ABB RAPID module: ecde059d.mod

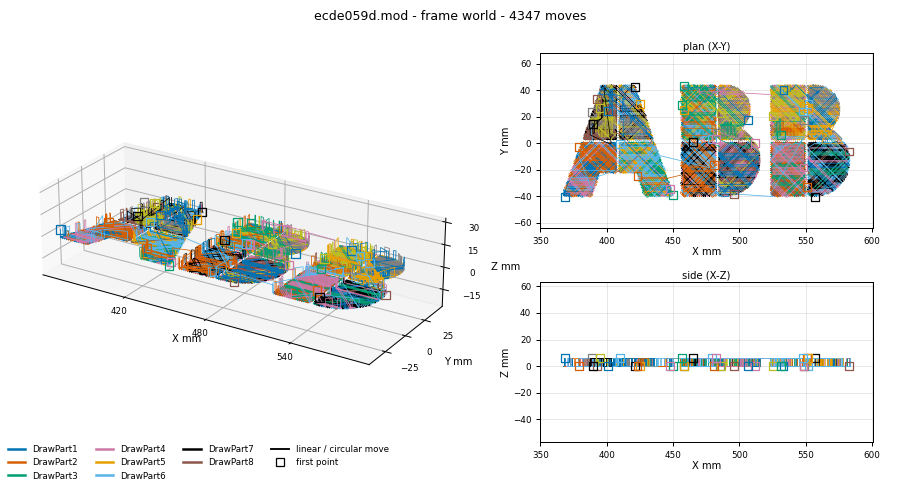
[picture p0: tool path of ecde059d.mod in frame world, 4347 of 4349 moves have a stored position in this frame; points joined in program order, loops and branches not executed]
MODULE ImageDraw
  ! Generated 2026-10-07 06:31 for ABB GoFa CRB 15000-5/0.95: 465 strokes
  ! Page 250 x 180 mm. Work object wPaper: Z points up, so pen-up is +Z and the tool uses orientation [0,1,0,0].
  PERS tooldata tPen:=[TRUE,[[0,0,120],[1,0,0,0]],[0.3,[0,0,60],[1,0,0,0],0,0,0]];
  PERS wobjdata wPaper:=[FALSE,TRUE,"",[[350,-90,0],[1,0,0,0]],[[0,0,0],[1,0,0,0]]];
  CONST robtarget pOrigin:=[[0,0,0],[0,1,0,0],[0,0,0,0],[9E9,9E9,9E9,9E9,9E9,9E9]];
  CONST jointtarget jHome:=[[0,0,0,0,30,0],[9E9,9E9,9E9,9E9,9E9,9E9]];
  CONST speeddata vTravel:=[250,200,5000,1000];

  PROC DrawImage()
    SingArea\Wrist;
    ConfL\Off;
    ConfJ\Off;
    MoveAbsJ jHome\NoEOffs,vTravel,fine,tPen;
    DrawPart1;
    DrawPart2;
    DrawPart3;
    DrawPart4;
    DrawPart5;
    DrawPart6;
    DrawPart7;
    DrawPart8;
    DrawPart9;
    DrawPart10;
    DrawPart11;
    DrawPart12;
    DrawPart13;
    DrawPart14;
    DrawPart15;
    DrawPart16;
    DrawPart17;
    DrawPart18;
    DrawPart19;
    DrawPart20;
    DrawPart21;
    DrawPart22;
    DrawPart23;
    DrawPart24;
    DrawPart25;
    DrawPart26;
    DrawPart27;
    DrawPart28;
    DrawPart29;
    DrawPart30;
    DrawPart31;
    DrawPart32;
    DrawPart33;
    DrawPart34;
    DrawPart35;
    DrawPart36;
    DrawPart37;
    MoveAbsJ jHome\NoEOffs,vTravel,fine,tPen;
  ENDPROC

  PROC DrawPart1()
    MoveL Offs(pOrigin,18.68,49.65,6.00),vTravel,z5,tPen\WObj:=wPaper;
    MoveL Offs(pOrigin,18.68,49.65,0.00),v60,z0,tPen\WObj:=wPaper;
    MoveL Offs(pOrigin,16.98,51.35,0.00),v40,z0,tPen\WObj:=wPaper;
    MoveL Offs(pOrigin,17.75,50.83,0.00),v40,z0,tPen\WObj:=wPaper;
    MoveL Offs(pOrigin,38.15,50.83,0.00),v40,z0,tPen\WObj:=wPaper;
    MoveL Offs(pOrigin,44.15,68.12,0.00),v40,z0,tPen\WObj:=wPaper;
    MoveL Offs(pOrigin,57.05,68.32,0.00),v40,z0,tPen\WObj:=wPaper;
    MoveL Offs(pOrigin,57.05,90.47,0.00),v40,z0,tPen\WObj:=wPaper;
    MoveL Offs(pOrigin,31.55,90.38,0.00),v40,z0,tPen\WObj:=wPaper;
    MoveL Offs(pOrigin,17.80,51.83,0.00),v40,z0,tPen\WObj:=wPaper;
    MoveL Offs(pOrigin,17.75,50.83,0.00),v40,z0,tPen\WObj:=wPaper;
    MoveL Offs(pOrigin,18.37,50.89,0.00),v40,z0,tPen\WObj:=wPaper;
    MoveL Offs(pOrigin,56.88,89.39,0.00),v40,z0,tPen\WObj:=wPaper;
    MoveL Offs(pOrigin,56.13,90.14,0.00),v40,z0,tPen\WObj:=wPaper;
    MoveL Offs(pOrigin,17.84,51.85,0.00),v40,z0,tPen\WObj:=wPaper;
    MoveL Offs(pOrigin,17.20,52.63,0.00),v40,z0,tPen\WObj:=wPaper;
    MoveL Offs(pOrigin,20.06,49.76,0.00),v40,z0,tPen\WObj:=wPaper;
    MoveL Offs(pOrigin,19.65,50.67,0.00),v40,z0,tPen\WObj:=wPaper;
    MoveL Offs(pOrigin,56.88,87.90,0.00),v40,z0,tPen\WObj:=wPaper;
    MoveL Offs(pOrigin,56.15,87.51,0.00),v40,z0,tPen\WObj:=wPaper;
    MoveL Offs(pOrigin,31.55,87.51,0.00),v40,z0,tPen\WObj:=wPaper;
    MoveL Offs(pOrigin,31.70,88.57,0.00),v40,z0,tPen\WObj:=wPaper;
    MoveL Offs(pOrigin,56.15,88.57,0.00),v40,fine,tPen\WObj:=wPaper;
    MoveL Offs(pOrigin,56.15,88.57,6.00),v60,z5,tPen\WObj:=wPaper;
    MoveL Offs(pOrigin,57.51,88.48,6.00),vTravel,z5,tPen\WObj:=wPaper;
    MoveL Offs(pOrigin,57.51,88.48,0.00),v60,z0,tPen\WObj:=wPaper;
    MoveL Offs(pOrigin,55.17,90.81,0.00),v40,z0,tPen\WObj:=wPaper;
    MoveL Offs(pOrigin,54.75,90.25,0.00),v40,z0,tPen\WObj:=wPaper;
    MoveL Offs(pOrigin,18.47,53.98,0.00),v40,z0,tPen\WObj:=wPaper;
    MoveL Offs(pOrigin,19.40,53.72,0.00),v40,z0,tPen\WObj:=wPaper;
    MoveL Offs(pOrigin,38.30,53.72,0.00),v40,z0,tPen\WObj:=wPaper;
    MoveL Offs(pOrigin,39.32,53.92,0.00),v40,z0,tPen\WObj:=wPaper;
    MoveL Offs(pOrigin,36.14,50.73,0.00),v40,fine,tPen\WObj:=wPaper;
    MoveL Offs(pOrigin,36.14,50.73,6.00),v60,z5,tPen\WObj:=wPaper;
    MoveL Offs(pOrigin,34.75,50.84,6.00),vTravel,z5,tPen\WObj:=wPaper;
    MoveL Offs(pOrigin,34.75,50.84,0.00),v60,z0,tPen\WObj:=wPaper;
    MoveL Offs(pOrigin,39.85,55.94,0.00),v40,z0,tPen\WObj:=wPaper;
    MoveL Offs(pOrigin,39.05,55.83,0.00),v40,z0,tPen\WObj:=wPaper;
    MoveL Offs(pOrigin,20.15,55.83,0.00),v40,z0,tPen\WObj:=wPaper;
    MoveL Offs(pOrigin,19.21,56.21,0.00),v40,z0,tPen\WObj:=wPaper;
    MoveL Offs(pOrigin,53.47,90.47,0.00),v40,z0,tPen\WObj:=wPaper;
    MoveL Offs(pOrigin,53.58,90.92,0.00),v40,z0,tPen\WObj:=wPaper;
    MoveL Offs(pOrigin,57.50,86.99,0.00),v40,z0,tPen\WObj:=wPaper;
    MoveL Offs(pOrigin,56.88,86.41,0.00),v40,z0,tPen\WObj:=wPaper;
    MoveL Offs(pOrigin,21.25,50.78,0.00),v40,z0,tPen\WObj:=wPaper;
    MoveL Offs(pOrigin,21.55,49.77,0.00),v40,z0,tPen\WObj:=wPaper;
    MoveL Offs(pOrigin,17.42,53.90,0.00),v40,fine,tPen\WObj:=wPaper;
    MoveL Offs(pOrigin,17.42,53.90,6.00),v60,z5,tPen\WObj:=wPaper;
    MoveL Offs(pOrigin,17.53,55.29,6.00),vTravel,z5,tPen\WObj:=wPaper;
    MoveL Offs(pOrigin,17.53,55.29,0.00),v60,z0,tPen\WObj:=wPaper;
    MoveL Offs(pOrigin,23.47,49.35,0.00),v40,fine,tPen\WObj:=wPaper;
    MoveL Offs(pOrigin,23.47,49.35,6.00),v60,z5,tPen\WObj:=wPaper;
    MoveL Offs(pOrigin,24.12,50.66,6.00),vTravel,z5,tPen\WObj:=wPaper;
    MoveL Offs(pOrigin,24.12,50.66,0.00),v60,z0,tPen\WObj:=wPaper;
    MoveL Offs(pOrigin,56.89,83.44,0.00),v40,z0,tPen\WObj:=wPaper;
    MoveL Offs(pOrigin,57.60,83.91,0.00),v40,z0,tPen\WObj:=wPaper;
    MoveL Offs(pOrigin,50.71,90.80,0.00),v40,z0,tPen\WObj:=wPaper;
    MoveL Offs(pOrigin,50.28,90.26,0.00),v40,z0,tPen\WObj:=wPaper;
    MoveL Offs(pOrigin,20.79,60.78,0.00),v40,z0,tPen\WObj:=wPaper;
    MoveL Offs(pOrigin,20.31,61.46,0.00),v40,z0,tPen\WObj:=wPaper;
    MoveL Offs(pOrigin,32.29,49.48,0.00),v40,fine,tPen\WObj:=wPaper;
    MoveL Offs(pOrigin,32.29,49.48,6.00),v60,z5,tPen\WObj:=wPaper;
    MoveL Offs(pOrigin,31.02,49.26,6.00),vTravel,z5,tPen\WObj:=wPaper;
    MoveL Offs(pOrigin,31.02,49.26,0.00),v60,z0,tPen\WObj:=wPaper;
    MoveL Offs(pOrigin,19.77,60.51,0.00),v40,z0,tPen\WObj:=wPaper;
    MoveL Offs(pOrigin,19.35,59.44,0.00),v40,z0,tPen\WObj:=wPaper;
    MoveL Offs(pOrigin,29.10,49.68,0.00),v40,z0,tPen\WObj:=wPaper;
    MoveL Offs(pOrigin,28.59,50.65,0.00),v40,z0,tPen\WObj:=wPaper;
    MoveL Offs(pOrigin,43.12,65.18,0.00),v40,z0,tPen\WObj:=wPaper;
    MoveL Offs(pOrigin,42.35,65.34,0.00),v40,z0,tPen\WObj:=wPaper;
    MoveL Offs(pOrigin,23.60,65.34,0.00),v40,z0,tPen\WObj:=wPaper;
    MoveL Offs(pOrigin,23.90,66.39,0.00),v40,z0,tPen\WObj:=wPaper;
    MoveL Offs(pOrigin,42.65,66.39,0.00),v40,z0,tPen\WObj:=wPaper;
    MoveL Offs(pOrigin,42.95,67.45,0.00),v40,z0,tPen\WObj:=wPaper;
    MoveL Offs(pOrigin,24.35,67.45,0.00),v40,z0,tPen\WObj:=wPaper;
    MoveL Offs(pOrigin,24.65,68.50,0.00),v40,z0,tPen\WObj:=wPaper;
    MoveL Offs(pOrigin,43.85,68.50,0.00),v40,fine,tPen\WObj:=wPaper;
    MoveL Offs(pOrigin,43.85,68.50,6.00),v60,z5,tPen\WObj:=wPaper;
    MoveL Offs(pOrigin,44.58,67.06,6.00),vTravel,z5,tPen\WObj:=wPaper;
    MoveL Offs(pOrigin,44.58,67.06,0.00),v60,z0,tPen\WObj:=wPaper;
    MoveL Offs(pOrigin,28.35,83.29,0.00),v40,z0,tPen\WObj:=wPaper;
    MoveL Offs(pOrigin,27.92,82.23,0.00),v40,z0,tPen\WObj:=wPaper;
    MoveL Offs(pOrigin,44.15,66.00,0.00),v40,fine,tPen\WObj:=wPaper;
    MoveL Offs(pOrigin,44.15,66.00,6.00),v60,z5,tPen\WObj:=wPaper;
    MoveL Offs(pOrigin,43.83,64.83,6.00),vTravel,z5,tPen\WObj:=wPaper;
    MoveL Offs(pOrigin,43.83,64.83,0.00),v60,z0,tPen\WObj:=wPaper;
    MoveL Offs(pOrigin,27.28,81.37,0.00),v40,z0,tPen\WObj:=wPaper;
    MoveL Offs(pOrigin,26.85,80.31,0.00),v40,z0,tPen\WObj:=wPaper;
    MoveL Offs(pOrigin,43.50,63.66,0.00),v40,z0,tPen\WObj:=wPaper;
    MoveL Offs(pOrigin,43.07,62.59,0.00),v40,z0,tPen\WObj:=wPaper;
    MoveL Offs(pOrigin,26.53,79.14,0.00),v40,z0,tPen\WObj:=wPaper;
    MoveL Offs(pOrigin,27.44,79.37,0.00),v40,z0,tPen\WObj:=wPaper;
    MoveL Offs(pOrigin,38.58,90.51,0.00),v40,z0,tPen\WObj:=wPaper;
    MoveL Offs(pOrigin,38.37,91.19,0.00),v40,z0,tPen\WObj:=wPaper;
    MoveL Offs(pOrigin,57.78,71.78,0.00),v40,z0,tPen\WObj:=wPaper;
    MoveL Offs(pOrigin,57.03,71.63,0.00),v40,z0,tPen\WObj:=wPaper;
    MoveL Offs(pOrigin,53.64,68.24,0.00),v40,z0,tPen\WObj:=wPaper;
    MoveL Offs(pOrigin,53.19,67.41,0.00),v40,z0,tPen\WObj:=wPaper;
    MoveL Offs(pOrigin,30.50,90.11,0.00),v40,z0,tPen\WObj:=wPaper;
    MoveL Offs(pOrigin,31.24,90.85,0.00),v40,z0,tPen\WObj:=wPaper;
    MoveL Offs(pOrigin,55.11,66.99,0.00),v40,fine,tPen\WObj:=wPaper;
    MoveL Offs(pOrigin,55.11,66.99,6.00),v60,z5,tPen\WObj:=wPaper;
    MoveL Offs(pOrigin,55.13,68.23,6.00),vTravel,z5,tPen\WObj:=wPaper;
    MoveL Offs(pOrigin,55.13,68.23,0.00),v60,z0,tPen\WObj:=wPaper;
    MoveL Offs(pOrigin,57.04,70.14,0.00),v40,z0,tPen\WObj:=wPaper;
    MoveL Offs(pOrigin,56.15,70.62,0.00),v40,z0,tPen\WObj:=wPaper;
    MoveL Offs(pOrigin,25.40,70.62,0.00),v40,z0,tPen\WObj:=wPaper;
    MoveL Offs(pOrigin,25.85,71.67,0.00),v40,z0,tPen\WObj:=wPaper;
    MoveL Offs(pOrigin,56.15,71.67,0.00),v40,z0,tPen\WObj:=wPaper;
    MoveL Offs(pOrigin,56.15,72.73,0.00),v40,z0,tPen\WObj:=wPaper;
    MoveL Offs(pOrigin,26.30,72.73,0.00),v40,z0,tPen\WObj:=wPaper;
    MoveL Offs(pOrigin,26.60,73.78,0.00),v40,z0,tPen\WObj:=wPaper;
    MoveL Offs(pOrigin,56.15,73.78,0.00),v40,z0,tPen\WObj:=wPaper;
    MoveL Offs(pOrigin,56.15,74.84,0.00),v40,z0,tPen\WObj:=wPaper;
    MoveL Offs(pOrigin,27.05,74.84,0.00),v40,z0,tPen\WObj:=wPaper;
    MoveL Offs(pOrigin,27.50,75.90,0.00),v40,z0,tPen\WObj:=wPaper;
    MoveL Offs(pOrigin,56.00,75.90,0.00),v40,z0,tPen\WObj:=wPaper;
    MoveL Offs(pOrigin,56.81,75.88,0.00),v40,z0,tPen\WObj:=wPaper;
    MoveL Offs(pOrigin,49.17,68.25,0.00),v40,z0,tPen\WObj:=wPaper;
    MoveL Offs(pOrigin,49.04,67.08,0.00),v40,z0,tPen\WObj:=wPaper;
  ENDPROC

  PROC DrawPart2()
    MoveL Offs(pOrigin,29.32,86.81,0.00),v40,z0,tPen\WObj:=wPaper;
    MoveL Offs(pOrigin,29.97,86.39,0.00),v40,z0,tPen\WObj:=wPaper;
    MoveL Offs(pOrigin,34.11,90.52,0.00),v40,z0,tPen\WObj:=wPaper;
    MoveL Offs(pOrigin,34.22,90.86,0.00),v40,z0,tPen\WObj:=wPaper;
    MoveL Offs(pOrigin,57.24,67.84,0.00),v40,z0,tPen\WObj:=wPaper;
    MoveL Offs(pOrigin,56.38,67.20,0.00),v40,z0,tPen\WObj:=wPaper;
    MoveL Offs(pOrigin,32.41,91.18,0.00),v40,z0,tPen\WObj:=wPaper;
    MoveL Offs(pOrigin,32.62,90.53,0.00),v40,z0,tPen\WObj:=wPaper;
    MoveL Offs(pOrigin,30.82,88.72,0.00),v40,z0,tPen\WObj:=wPaper;
    MoveL Offs(pOrigin,30.17,88.94,0.00),v40,z0,tPen\WObj:=wPaper;
    MoveL Offs(pOrigin,51.70,67.40,0.00),v40,z0,tPen\WObj:=wPaper;
    MoveL Offs(pOrigin,52.26,68.35,0.00),v40,z0,tPen\WObj:=wPaper;
    MoveL Offs(pOrigin,57.03,73.12,0.00),v40,z0,tPen\WObj:=wPaper;
    MoveL Offs(pOrigin,57.78,73.27,0.00),v40,z0,tPen\WObj:=wPaper;
    MoveL Offs(pOrigin,40.18,90.88,0.00),v40,z0,tPen\WObj:=wPaper;
    MoveL Offs(pOrigin,40.07,90.50,0.00),v40,z0,tPen\WObj:=wPaper;
    MoveL Offs(pOrigin,26.81,77.25,0.00),v40,z0,tPen\WObj:=wPaper;
    MoveL Offs(pOrigin,27.80,76.95,0.00),v40,z0,tPen\WObj:=wPaper;
    MoveL Offs(pOrigin,56.00,76.95,0.00),v40,z0,tPen\WObj:=wPaper;
    MoveL Offs(pOrigin,56.80,77.37,0.00),v40,z0,tPen\WObj:=wPaper;
    MoveL Offs(pOrigin,47.68,68.25,0.00),v40,z0,tPen\WObj:=wPaper;
    MoveL Offs(pOrigin,47.34,67.28,0.00),v40,z0,tPen\WObj:=wPaper;
    MoveL Offs(pOrigin,28.99,85.63,0.00),v40,fine,tPen\WObj:=wPaper;
    MoveL Offs(pOrigin,28.99,85.63,6.00),v60,z5,tPen\WObj:=wPaper;
    MoveL Offs(pOrigin,28.67,84.46,6.00),vTravel,z5,tPen\WObj:=wPaper;
    MoveL Offs(pOrigin,28.67,84.46,0.00),v60,z0,tPen\WObj:=wPaper;
    MoveL Offs(pOrigin,45.75,67.39,0.00),v40,z0,tPen\WObj:=wPaper;
    MoveL Offs(pOrigin,46.19,68.26,0.00),v40,z0,tPen\WObj:=wPaper;
    MoveL Offs(pOrigin,56.91,78.97,0.00),v40,z0,tPen\WObj:=wPaper;
    MoveL Offs(pOrigin,57.48,79.55,0.00),v40,z0,tPen\WObj:=wPaper;
    MoveL Offs(pOrigin,46.13,90.90,0.00),v40,z0,tPen\WObj:=wPaper;
    MoveL Offs(pOrigin,46.02,90.49,0.00),v40,z0,tPen\WObj:=wPaper;
    MoveL Offs(pOrigin,23.22,67.68,0.00),v40,z0,tPen\WObj:=wPaper;
    MoveL Offs(pOrigin,22.46,68.28,0.00),v40,z0,tPen\WObj:=wPaper;
    MoveL Offs(pOrigin,39.43,51.31,0.00),v40,z0,tPen\WObj:=wPaper;
    MoveL Offs(pOrigin,38.89,50.35,0.00),v40,z0,tPen\WObj:=wPaper;
    MoveL Offs(pOrigin,22.03,67.21,0.00),v40,z0,tPen\WObj:=wPaper;
    MoveL Offs(pOrigin,21.49,66.25,0.00),v40,z0,tPen\WObj:=wPaper;
    MoveL Offs(pOrigin,38.25,49.50,0.00),v40,fine,tPen\WObj:=wPaper;
    MoveL Offs(pOrigin,38.25,49.50,6.00),v60,z5,tPen\WObj:=wPaper;
    MoveL Offs(pOrigin,36.76,49.49,6.00),vTravel,z5,tPen\WObj:=wPaper;
    MoveL Offs(pOrigin,36.76,49.49,0.00),v60,z0,tPen\WObj:=wPaper;
    MoveL Offs(pOrigin,21.06,65.19,0.00),v40,fine,tPen\WObj:=wPaper;
    MoveL Offs(pOrigin,21.06,65.19,6.00),v60,z5,tPen\WObj:=wPaper;
    MoveL Offs(pOrigin,22.27,65.24,6.00),vTravel,z5,tPen\WObj:=wPaper;
    MoveL Offs(pOrigin,22.27,65.24,0.00),v60,z0,tPen\WObj:=wPaper;
    MoveL Offs(pOrigin,47.30,90.27,0.00),v40,z0,tPen\WObj:=wPaper;
    MoveL Offs(pOrigin,47.73,90.79,0.00),v40,z0,tPen\WObj:=wPaper;
    MoveL Offs(pOrigin,57.49,81.04,0.00),v40,z0,tPen\WObj:=wPaper;
    MoveL Offs(pOrigin,56.90,80.46,0.00),v40,z0,tPen\WObj:=wPaper;
    MoveL Offs(pOrigin,27.10,50.65,0.00),v40,z0,tPen\WObj:=wPaper;
    MoveL Offs(pOrigin,27.51,49.78,0.00),v40,z0,tPen\WObj:=wPaper;
    MoveL Offs(pOrigin,19.02,58.27,0.00),v40,z0,tPen\WObj:=wPaper;
    MoveL Offs(pOrigin,19.95,58.44,0.00),v40,z0,tPen\WObj:=wPaper;
    MoveL Offs(pOrigin,51.98,90.47,0.00),v40,z0,tPen\WObj:=wPaper;
    MoveL Offs(pOrigin,52.09,90.91,0.00),v40,z0,tPen\WObj:=wPaper;
    MoveL Offs(pOrigin,57.50,85.50,0.00),v40,z0,tPen\WObj:=wPaper;
    MoveL Offs(pOrigin,56.89,84.93,0.00),v40,z0,tPen\WObj:=wPaper;
    MoveL Offs(pOrigin,22.63,50.67,0.00),v40,fine,tPen\WObj:=wPaper;
    MoveL Offs(pOrigin,22.63,50.67,6.00),v60,z5,tPen\WObj:=wPaper;
    MoveL Offs(pOrigin,24.95,49.35,6.00),vTravel,z5,tPen\WObj:=wPaper;
    MoveL Offs(pOrigin,24.95,49.35,0.00),v60,z0,tPen\WObj:=wPaper;
    MoveL Offs(pOrigin,17.95,56.35,0.00),v40,z0,tPen\WObj:=wPaper;
    MoveL Offs(pOrigin,18.59,57.20,0.00),v40,z0,tPen\WObj:=wPaper;
    MoveL Offs(pOrigin,26.13,49.67,0.00),v40,z0,tPen\WObj:=wPaper;
    MoveL Offs(pOrigin,25.61,50.66,0.00),v40,z0,tPen\WObj:=wPaper;
    MoveL Offs(pOrigin,56.79,81.84,0.00),v40,z0,tPen\WObj:=wPaper;
    MoveL Offs(pOrigin,56.00,82.23,0.00),v40,z0,tPen\WObj:=wPaper;
    MoveL Offs(pOrigin,29.60,82.23,0.00),v40,z0,tPen\WObj:=wPaper;
    MoveL Offs(pOrigin,29.30,81.18,0.00),v40,z0,tPen\WObj:=wPaper;
    MoveL Offs(pOrigin,56.00,81.18,0.00),v40,z0,tPen\WObj:=wPaper;
    MoveL Offs(pOrigin,56.00,80.12,0.00),v40,z0,tPen\WObj:=wPaper;
    MoveL Offs(pOrigin,28.85,80.12,0.00),v40,z0,tPen\WObj:=wPaper;
    MoveL Offs(pOrigin,28.55,79.06,0.00),v40,z0,tPen\WObj:=wPaper;
    MoveL Offs(pOrigin,55.85,79.06,0.00),v40,z0,tPen\WObj:=wPaper;
    MoveL Offs(pOrigin,55.85,78.01,0.00),v40,z0,tPen\WObj:=wPaper;
    MoveL Offs(pOrigin,28.10,78.01,0.00),v40,fine,tPen\WObj:=wPaper;
    MoveL Offs(pOrigin,28.10,78.01,6.00),v60,z5,tPen\WObj:=wPaper;
    MoveL Offs(pOrigin,26.10,78.07,6.00),vTravel,z5,tPen\WObj:=wPaper;
    MoveL Offs(pOrigin,26.10,78.07,0.00),v60,z0,tPen\WObj:=wPaper;
    MoveL Offs(pOrigin,42.75,61.42,0.00),v40,fine,tPen\WObj:=wPaper;
    MoveL Offs(pOrigin,42.75,61.42,6.00),v60,z5,tPen\WObj:=wPaper;
    MoveL Offs(pOrigin,42.64,60.04,6.00),vTravel,z5,tPen\WObj:=wPaper;
    MoveL Offs(pOrigin,42.64,60.04,0.00),v60,z0,tPen\WObj:=wPaper;
    MoveL Offs(pOrigin,25.67,77.01,0.00),v40,z0,tPen\WObj:=wPaper;
    MoveL Offs(pOrigin,25.14,76.05,0.00),v40,z0,tPen\WObj:=wPaper;
    MoveL Offs(pOrigin,42.32,58.87,0.00),v40,z0,tPen\WObj:=wPaper;
    MoveL Offs(pOrigin,41.78,57.91,0.00),v40,z0,tPen\WObj:=wPaper;
    MoveL Offs(pOrigin,24.92,74.77,0.00),v40,z0,tPen\WObj:=wPaper;
    MoveL Offs(pOrigin,25.86,74.80,0.00),v40,z0,tPen\WObj:=wPaper;
    MoveL Offs(pOrigin,41.34,90.29,0.00),v40,z0,tPen\WObj:=wPaper;
    MoveL Offs(pOrigin,41.77,90.78,0.00),v40,z0,tPen\WObj:=wPaper;
    MoveL Offs(pOrigin,57.79,74.76,0.00),v40,z0,tPen\WObj:=wPaper;
    MoveL Offs(pOrigin,57.02,74.61,0.00),v40,z0,tPen\WObj:=wPaper;
    MoveL Offs(pOrigin,50.66,68.24,0.00),v40,z0,tPen\WObj:=wPaper;
    MoveL Offs(pOrigin,50.32,67.29,0.00),v40,z0,tPen\WObj:=wPaper;
    MoveL Offs(pOrigin,29.74,87.87,0.00),v40,fine,tPen\WObj:=wPaper;
    MoveL Offs(pOrigin,29.74,87.87,6.00),v60,z5,tPen\WObj:=wPaper;
    MoveL Offs(pOrigin,31.10,86.46,6.00),vTravel,z5,tPen\WObj:=wPaper;
    MoveL Offs(pOrigin,31.10,86.46,0.00),v60,z0,tPen\WObj:=wPaper;
    MoveL Offs(pOrigin,56.00,86.46,0.00),v40,z0,tPen\WObj:=wPaper;
    MoveL Offs(pOrigin,56.00,85.40,0.00),v40,z0,tPen\WObj:=wPaper;
    MoveL Offs(pOrigin,30.80,85.40,0.00),v40,z0,tPen\WObj:=wPaper;
    MoveL Offs(pOrigin,30.50,84.34,0.00),v40,z0,tPen\WObj:=wPaper;
    MoveL Offs(pOrigin,56.00,84.34,0.00),v40,z0,tPen\WObj:=wPaper;
    MoveL Offs(pOrigin,56.00,83.29,0.00),v40,z0,tPen\WObj:=wPaper;
    MoveL Offs(pOrigin,30.05,83.29,0.00),v40,fine,tPen\WObj:=wPaper;
    MoveL Offs(pOrigin,30.05,83.29,6.00),v60,z5,tPen\WObj:=wPaper;
    MoveL Offs(pOrigin,29.34,84.26,6.00),vTravel,z5,tPen\WObj:=wPaper;
    MoveL Offs(pOrigin,29.34,84.26,0.00),v60,z0,tPen\WObj:=wPaper;
    MoveL Offs(pOrigin,35.60,90.52,0.00),v40,z0,tPen\WObj:=wPaper;
    MoveL Offs(pOrigin,35.71,90.87,0.00),v40,z0,tPen\WObj:=wPaper;
    MoveL Offs(pOrigin,57.88,68.70,0.00),v40,fine,tPen\WObj:=wPaper;
    MoveL Offs(pOrigin,57.88,68.70,6.00),v60,z5,tPen\WObj:=wPaper;
    MoveL Offs(pOrigin,59.45,68.78,6.00),vTravel,z5,tPen\WObj:=wPaper;
    MoveL Offs(pOrigin,59.45,68.78,0.00),v60,z0,tPen\WObj:=wPaper;
    MoveL Offs(pOrigin,59.75,68.22,0.00),v40,z0,tPen\WObj:=wPaper;
    MoveL Offs(pOrigin,73.05,68.12,0.00),v40,z0,tPen\WObj:=wPaper;
    MoveL Offs(pOrigin,79.10,50.83,0.00),v40,z0,tPen\WObj:=wPaper;
    MoveL Offs(pOrigin,99.05,50.62,0.00),v40,z0,tPen\WObj:=wPaper;
  ENDPROC

  PROC DrawPart3()
    MoveL Offs(pOrigin,99.60,50.92,0.00),v40,z0,tPen\WObj:=wPaper;
    MoveL Offs(pOrigin,85.65,90.47,0.00),v40,z0,tPen\WObj:=wPaper;
    MoveL Offs(pOrigin,59.65,90.38,0.00),v40,z0,tPen\WObj:=wPaper;
    MoveL Offs(pOrigin,59.45,68.78,0.00),v40,z0,tPen\WObj:=wPaper;
    MoveL Offs(pOrigin,60.02,68.64,0.00),v40,z0,tPen\WObj:=wPaper;
    MoveL Offs(pOrigin,81.98,90.60,0.00),v40,fine,tPen\WObj:=wPaper;
    MoveL Offs(pOrigin,81.98,90.60,6.00),v60,z5,tPen\WObj:=wPaper;
    MoveL Offs(pOrigin,80.70,90.81,6.00),vTravel,z5,tPen\WObj:=wPaper;
    MoveL Offs(pOrigin,80.70,90.81,0.00),v60,z0,tPen\WObj:=wPaper;
    MoveL Offs(pOrigin,59.49,69.60,0.00),v40,z0,tPen\WObj:=wPaper;
    MoveL Offs(pOrigin,60.65,69.56,0.00),v40,z0,tPen\WObj:=wPaper;
    MoveL Offs(pOrigin,92.15,69.56,0.00),v40,z0,tPen\WObj:=wPaper;
    MoveL Offs(pOrigin,92.88,70.14,0.00),v40,z0,tPen\WObj:=wPaper;
    MoveL Offs(pOrigin,77.50,54.76,0.00),v40,z0,tPen\WObj:=wPaper;
    MoveL Offs(pOrigin,76.77,54.29,0.00),v40,z0,tPen\WObj:=wPaper;
    MoveL Offs(pOrigin,81.54,49.51,0.00),v40,fine,tPen\WObj:=wPaper;
    MoveL Offs(pOrigin,81.54,49.51,6.00),v60,z5,tPen\WObj:=wPaper;
    MoveL Offs(pOrigin,80.37,49.19,6.00),vTravel,z5,tPen\WObj:=wPaper;
    MoveL Offs(pOrigin,80.37,49.19,0.00),v60,z0,tPen\WObj:=wPaper;
    MoveL Offs(pOrigin,76.77,52.80,0.00),v40,fine,tPen\WObj:=wPaper;
    MoveL Offs(pOrigin,76.77,52.80,6.00),v60,z5,tPen\WObj:=wPaper;
    MoveL Offs(pOrigin,77.83,53.59,6.00),vTravel,z5,tPen\WObj:=wPaper;
    MoveL Offs(pOrigin,77.83,53.59,0.00),v60,z0,tPen\WObj:=wPaper;
    MoveL Offs(pOrigin,93.31,69.08,0.00),v40,z0,tPen\WObj:=wPaper;
    MoveL Offs(pOrigin,92.45,68.50,0.00),v40,z0,tPen\WObj:=wPaper;
    MoveL Offs(pOrigin,73.40,68.50,0.00),v40,z0,tPen\WObj:=wPaper;
    MoveL Offs(pOrigin,72.79,67.97,0.00),v40,z0,tPen\WObj:=wPaper;
    MoveL Offs(pOrigin,88.17,83.35,0.00),v40,z0,tPen\WObj:=wPaper;
    MoveL Offs(pOrigin,87.20,83.29,0.00),v40,z0,tPen\WObj:=wPaper;
    MoveL Offs(pOrigin,60.65,83.29,0.00),v40,z0,tPen\WObj:=wPaper;
    MoveL Offs(pOrigin,59.77,83.32,0.00),v40,z0,tPen\WObj:=wPaper;
    MoveL Offs(pOrigin,66.98,90.53,0.00),v40,z0,tPen\WObj:=wPaper;
    MoveL Offs(pOrigin,66.66,91.27,0.00),v40,z0,tPen\WObj:=wPaper;
    MoveL Offs(pOrigin,97.53,60.41,0.00),v40,z0,tPen\WObj:=wPaper;
    MoveL Offs(pOrigin,96.42,60.24,0.00),v40,z0,tPen\WObj:=wPaper;
    MoveL Offs(pOrigin,86.88,50.70,0.00),v40,fine,tPen\WObj:=wPaper;
    MoveL Offs(pOrigin,86.88,50.70,6.00),v60,z5,tPen\WObj:=wPaper;
    MoveL Offs(pOrigin,85.90,49.63,6.00),vTravel,z5,tPen\WObj:=wPaper;
    MoveL Offs(pOrigin,85.90,49.63,0.00),v60,z0,tPen\WObj:=wPaper;
    MoveL Offs(pOrigin,73.92,61.62,0.00),v40,fine,tPen\WObj:=wPaper;
    MoveL Offs(pOrigin,73.92,61.62,6.00),v60,z5,tPen\WObj:=wPaper;
    MoveL Offs(pOrigin,74.82,62.54,6.00),vTravel,z5,tPen\WObj:=wPaper;
    MoveL Offs(pOrigin,74.82,62.54,0.00),v60,z0,tPen\WObj:=wPaper;
    MoveL Offs(pOrigin,90.10,77.81,0.00),v40,z0,tPen\WObj:=wPaper;
    MoveL Offs(pOrigin,89.45,76.95,0.00),v40,z0,tPen\WObj:=wPaper;
    MoveL Offs(pOrigin,60.50,76.95,0.00),v40,z0,tPen\WObj:=wPaper;
    MoveL Offs(pOrigin,59.68,77.26,0.00),v40,z0,tPen\WObj:=wPaper;
    MoveL Offs(pOrigin,73.04,90.62,0.00),v40,fine,tPen\WObj:=wPaper;
    MoveL Offs(pOrigin,73.04,90.62,6.00),v60,z5,tPen\WObj:=wPaper;
    MoveL Offs(pOrigin,74.53,90.62,6.00),vTravel,z5,tPen\WObj:=wPaper;
    MoveL Offs(pOrigin,74.53,90.62,0.00),v60,z0,tPen\WObj:=wPaper;
    MoveL Offs(pOrigin,59.68,75.77,0.00),v40,z0,tPen\WObj:=wPaper;
    MoveL Offs(pOrigin,60.50,75.90,0.00),v40,z0,tPen\WObj:=wPaper;
    MoveL Offs(pOrigin,89.75,75.90,0.00),v40,z0,tPen\WObj:=wPaper;
    MoveL Offs(pOrigin,90.05,74.84,0.00),v40,z0,tPen\WObj:=wPaper;
    MoveL Offs(pOrigin,60.50,74.84,0.00),v40,z0,tPen\WObj:=wPaper;
    MoveL Offs(pOrigin,59.68,74.28,0.00),v40,z0,tPen\WObj:=wPaper;
    MoveL Offs(pOrigin,75.91,90.51,0.00),v40,z0,tPen\WObj:=wPaper;
    MoveL Offs(pOrigin,75.70,91.19,0.00),v40,z0,tPen\WObj:=wPaper;
    MoveL Offs(pOrigin,92.04,74.86,0.00),v40,z0,tPen\WObj:=wPaper;
    MoveL Offs(pOrigin,91.17,74.40,0.00),v40,z0,tPen\WObj:=wPaper;
    MoveL Offs(pOrigin,76.00,59.24,0.00),v40,z0,tPen\WObj:=wPaper;
    MoveL Offs(pOrigin,75.08,58.96,0.00),v40,z0,tPen\WObj:=wPaper;
    MoveL Offs(pOrigin,84.31,49.73,0.00),v40,z0,tPen\WObj:=wPaper;
    MoveL Offs(pOrigin,83.90,50.70,0.00),v40,z0,tPen\WObj:=wPaper;
    MoveL Offs(pOrigin,95.56,62.37,0.00),v40,z0,tPen\WObj:=wPaper;
    MoveL Offs(pOrigin,94.85,62.17,0.00),v40,z0,tPen\WObj:=wPaper;
    MoveL Offs(pOrigin,75.95,62.17,0.00),v40,z0,tPen\WObj:=wPaper;
    MoveL Offs(pOrigin,75.36,61.58,0.00),v40,z0,tPen\WObj:=wPaper;
    MoveL Offs(pOrigin,90.52,76.75,0.00),v40,z0,tPen\WObj:=wPaper;
    MoveL Offs(pOrigin,91.09,77.30,0.00),v40,z0,tPen\WObj:=wPaper;
    MoveL Offs(pOrigin,77.19,91.20,0.00),v40,z0,tPen\WObj:=wPaper;
    MoveL Offs(pOrigin,77.51,90.61,0.00),v40,z0,tPen\WObj:=wPaper;
    MoveL Offs(pOrigin,59.69,72.79,0.00),v40,z0,tPen\WObj:=wPaper;
    MoveL Offs(pOrigin,60.50,72.73,0.00),v40,z0,tPen\WObj:=wPaper;
    MoveL Offs(pOrigin,90.95,72.73,0.00),v40,z0,tPen\WObj:=wPaper;
    MoveL Offs(pOrigin,91.60,73.34,0.00),v40,z0,tPen\WObj:=wPaper;
    MoveL Offs(pOrigin,76.32,58.07,0.00),v40,z0,tPen\WObj:=wPaper;
    MoveL Offs(pOrigin,77.45,57.94,0.00),v40,z0,tPen\WObj:=wPaper;
    MoveL Offs(pOrigin,96.35,57.94,0.00),v40,z0,tPen\WObj:=wPaper;
    MoveL Offs(pOrigin,97.28,58.11,0.00),v40,z0,tPen\WObj:=wPaper;
    MoveL Offs(pOrigin,89.85,50.69,0.00),v40,z0,tPen\WObj:=wPaper;
    MoveL Offs(pOrigin,90.27,49.75,0.00),v40,z0,tPen\WObj:=wPaper;
    MoveL Offs(pOrigin,59.08,80.93,0.00),v40,z0,tPen\WObj:=wPaper;
    MoveL Offs(pOrigin,59.77,80.34,0.00),v40,z0,tPen\WObj:=wPaper;
    MoveL Offs(pOrigin,69.96,90.53,0.00),v40,z0,tPen\WObj:=wPaper;
    MoveL Offs(pOrigin,69.85,91.07,0.00),v40,z0,tPen\WObj:=wPaper;
    MoveL Offs(pOrigin,95.10,65.83,0.00),v40,z0,tPen\WObj:=wPaper;
    MoveL Offs(pOrigin,94.39,65.67,0.00),v40,z0,tPen\WObj:=wPaper;
    MoveL Offs(pOrigin,79.54,50.82,0.00),v40,z0,tPen\WObj:=wPaper;
    MoveL Offs(pOrigin,79.85,51.61,0.00),v40,z0,tPen\WObj:=wPaper;
    MoveL Offs(pOrigin,98.00,51.61,0.00),v40,z0,tPen\WObj:=wPaper;
    MoveL Offs(pOrigin,98.15,52.66,0.00),v40,z0,tPen\WObj:=wPaper;
    MoveL Offs(pOrigin,79.10,52.66,0.00),v40,z0,tPen\WObj:=wPaper;
    MoveL Offs(pOrigin,78.25,52.53,0.00),v40,z0,tPen\WObj:=wPaper;
    MoveL Offs(pOrigin,93.63,67.91,0.00),v40,z0,tPen\WObj:=wPaper;
    MoveL Offs(pOrigin,92.90,67.45,0.00),v40,z0,tPen\WObj:=wPaper;
    MoveL Offs(pOrigin,74.30,67.45,0.00),v40,z0,tPen\WObj:=wPaper;
    MoveL Offs(pOrigin,73.43,67.12,0.00),v40,z0,tPen\WObj:=wPaper;
    MoveL Offs(pOrigin,88.59,82.28,0.00),v40,z0,tPen\WObj:=wPaper;
    MoveL Offs(pOrigin,87.65,82.23,0.00),v40,z0,tPen\WObj:=wPaper;
    MoveL Offs(pOrigin,60.65,82.23,0.00),v40,z0,tPen\WObj:=wPaper;
    MoveL Offs(pOrigin,59.88,81.94,0.00),v40,z0,tPen\WObj:=wPaper;
    MoveL Offs(pOrigin,68.36,90.42,0.00),v40,z0,tPen\WObj:=wPaper;
    MoveL Offs(pOrigin,68.36,91.06,0.00),v40,z0,tPen\WObj:=wPaper;
    MoveL Offs(pOrigin,96.26,63.17,0.00),v40,z0,tPen\WObj:=wPaper;
    MoveL Offs(pOrigin,95.24,63.54,0.00),v40,z0,tPen\WObj:=wPaper;
    MoveL Offs(pOrigin,82.41,50.71,0.00),v40,z0,tPen\WObj:=wPaper;
    MoveL Offs(pOrigin,82.82,49.73,0.00),v40,z0,tPen\WObj:=wPaper;
    MoveL Offs(pOrigin,75.82,56.73,0.00),v40,z0,tPen\WObj:=wPaper;
    MoveL Offs(pOrigin,76.75,57.00,0.00),v40,z0,tPen\WObj:=wPaper;
    MoveL Offs(pOrigin,92.03,72.27,0.00),v40,z0,tPen\WObj:=wPaper;
    MoveL Offs(pOrigin,91.40,71.67,0.00),v40,z0,tPen\WObj:=wPaper;
    MoveL Offs(pOrigin,60.50,71.67,0.00),v40,z0,tPen\WObj:=wPaper;
    MoveL Offs(pOrigin,60.50,70.62,0.00),v40,z0,tPen\WObj:=wPaper;
    MoveL Offs(pOrigin,91.70,70.62,0.00),v40,z0,tPen\WObj:=wPaper;
    MoveL Offs(pOrigin,92.35,71.10,0.00),v40,z0,tPen\WObj:=wPaper;
    MoveL Offs(pOrigin,77.18,55.94,0.00),v40,z0,tPen\WObj:=wPaper;
    MoveL Offs(pOrigin,78.20,55.83,0.00),v40,z0,tPen\WObj:=wPaper;
    MoveL Offs(pOrigin,97.10,55.83,0.00),v40,z0,tPen\WObj:=wPaper;
  ENDPROC

  PROC DrawPart4()
    MoveL Offs(pOrigin,97.92,55.77,0.00),v40,z0,tPen\WObj:=wPaper;
    MoveL Offs(pOrigin,92.83,50.68,0.00),v40,fine,tPen\WObj:=wPaper;
    MoveL Offs(pOrigin,92.83,50.68,6.00),v60,z5,tPen\WObj:=wPaper;
    MoveL Offs(pOrigin,93.46,49.55,6.00),vTravel,z5,tPen\WObj:=wPaper;
    MoveL Offs(pOrigin,93.46,49.55,0.00),v60,z0,tPen\WObj:=wPaper;
    MoveL Offs(pOrigin,58.98,84.02,0.00),v40,z0,tPen\WObj:=wPaper;
    MoveL Offs(pOrigin,59.76,84.81,0.00),v40,z0,tPen\WObj:=wPaper;
    MoveL Offs(pOrigin,65.38,90.43,0.00),v40,z0,tPen\WObj:=wPaper;
    MoveL Offs(pOrigin,65.28,91.16,0.00),v40,z0,tPen\WObj:=wPaper;
    MoveL Offs(pOrigin,98.48,57.96,0.00),v40,fine,tPen\WObj:=wPaper;
    MoveL Offs(pOrigin,98.48,57.96,6.00),v60,z5,tPen\WObj:=wPaper;
    MoveL Offs(pOrigin,97.49,56.84,6.00),vTravel,z5,tPen\WObj:=wPaper;
    MoveL Offs(pOrigin,97.49,56.84,0.00),v60,z0,tPen\WObj:=wPaper;
    MoveL Offs(pOrigin,91.34,50.68,0.00),v40,z0,tPen\WObj:=wPaper;
    MoveL Offs(pOrigin,91.75,49.75,0.00),v40,z0,tPen\WObj:=wPaper;
    MoveL Offs(pOrigin,58.98,82.53,0.00),v40,fine,tPen\WObj:=wPaper;
    MoveL Offs(pOrigin,58.98,82.53,6.00),v60,z5,tPen\WObj:=wPaper;
    MoveL Offs(pOrigin,57.49,82.52,6.00),vTravel,z5,tPen\WObj:=wPaper;
    MoveL Offs(pOrigin,57.49,82.52,0.00),v60,z0,tPen\WObj:=wPaper;
    MoveL Offs(pOrigin,49.22,90.80,0.00),v40,z0,tPen\WObj:=wPaper;
    MoveL Offs(pOrigin,48.79,90.27,0.00),v40,z0,tPen\WObj:=wPaper;
    MoveL Offs(pOrigin,21.85,63.33,0.00),v40,z0,tPen\WObj:=wPaper;
    MoveL Offs(pOrigin,22.70,63.22,0.00),v40,z0,tPen\WObj:=wPaper;
    MoveL Offs(pOrigin,41.60,63.22,0.00),v40,z0,tPen\WObj:=wPaper;
    MoveL Offs(pOrigin,42.17,62.74,0.00),v40,z0,tPen\WObj:=wPaper;
    MoveL Offs(pOrigin,30.18,50.75,0.00),v40,fine,tPen\WObj:=wPaper;
    MoveL Offs(pOrigin,30.18,50.75,6.00),v60,z5,tPen\WObj:=wPaper;
    MoveL Offs(pOrigin,31.67,50.75,6.00),vTravel,z5,tPen\WObj:=wPaper;
    MoveL Offs(pOrigin,31.67,50.75,0.00),v60,z0,tPen\WObj:=wPaper;
    MoveL Offs(pOrigin,41.53,60.61,0.00),v40,z0,tPen\WObj:=wPaper;
    MoveL Offs(pOrigin,40.85,61.11,0.00),v40,z0,tPen\WObj:=wPaper;
    MoveL Offs(pOrigin,21.95,61.11,0.00),v40,z0,tPen\WObj:=wPaper;
    MoveL Offs(pOrigin,21.65,60.06,0.00),v40,z0,tPen\WObj:=wPaper;
    MoveL Offs(pOrigin,40.55,60.06,0.00),v40,z0,tPen\WObj:=wPaper;
    MoveL Offs(pOrigin,40.25,59.00,0.00),v40,z0,tPen\WObj:=wPaper;
    MoveL Offs(pOrigin,21.20,59.00,0.00),v40,z0,tPen\WObj:=wPaper;
    MoveL Offs(pOrigin,20.90,57.94,0.00),v40,z0,tPen\WObj:=wPaper;
    MoveL Offs(pOrigin,39.80,57.94,0.00),v40,z0,tPen\WObj:=wPaper;
    MoveL Offs(pOrigin,40.80,58.38,0.00),v40,z0,tPen\WObj:=wPaper;
    MoveL Offs(pOrigin,33.16,50.74,0.00),v40,z0,tPen\WObj:=wPaper;
    MoveL Offs(pOrigin,33.57,49.69,0.00),v40,z0,tPen\WObj:=wPaper;
    MoveL Offs(pOrigin,20.74,62.53,0.00),v40,fine,tPen\WObj:=wPaper;
    MoveL Offs(pOrigin,20.74,62.53,6.00),v60,z5,tPen\WObj:=wPaper;
    MoveL Offs(pOrigin,21.06,63.70,6.00),vTravel,z5,tPen\WObj:=wPaper;
    MoveL Offs(pOrigin,21.06,63.70,0.00),v60,z0,tPen\WObj:=wPaper;
    MoveL Offs(pOrigin,35.06,49.70,0.00),v40,fine,tPen\WObj:=wPaper;
    MoveL Offs(pOrigin,35.06,49.70,6.00),v60,z5,tPen\WObj:=wPaper;
    MoveL Offs(pOrigin,37.25,51.61,6.00),vTravel,z5,tPen\WObj:=wPaper;
    MoveL Offs(pOrigin,37.25,51.61,0.00),v60,z0,tPen\WObj:=wPaper;
    MoveL Offs(pOrigin,19.10,51.61,0.00),v40,z0,tPen\WObj:=wPaper;
    MoveL Offs(pOrigin,19.10,52.66,0.00),v40,z0,tPen\WObj:=wPaper;
    MoveL Offs(pOrigin,38.00,52.66,0.00),v40,fine,tPen\WObj:=wPaper;
    MoveL Offs(pOrigin,38.00,52.66,6.00),v60,z5,tPen\WObj:=wPaper;
    MoveL Offs(pOrigin,39.85,52.37,6.00),vTravel,z5,tPen\WObj:=wPaper;
    MoveL Offs(pOrigin,39.85,52.37,0.00),v60,z0,tPen\WObj:=wPaper;
    MoveL Offs(pOrigin,22.88,69.34,0.00),v40,fine,tPen\WObj:=wPaper;
    MoveL Offs(pOrigin,22.88,69.34,6.00),v60,z5,tPen\WObj:=wPaper;
    MoveL Offs(pOrigin,23.21,70.51,6.00),vTravel,z5,tPen\WObj:=wPaper;
    MoveL Offs(pOrigin,23.21,70.51,0.00),v60,z0,tPen\WObj:=wPaper;
    MoveL Offs(pOrigin,40.18,53.54,0.00),v40,fine,tPen\WObj:=wPaper;
    MoveL Offs(pOrigin,40.18,53.54,6.00),v60,z5,tPen\WObj:=wPaper;
    MoveL Offs(pOrigin,40.50,54.71,6.00),vTravel,z5,tPen\WObj:=wPaper;
    MoveL Offs(pOrigin,40.50,54.71,0.00),v60,z0,tPen\WObj:=wPaper;
    MoveL Offs(pOrigin,23.74,71.47,0.00),v40,z0,tPen\WObj:=wPaper;
    MoveL Offs(pOrigin,24.28,72.43,0.00),v40,z0,tPen\WObj:=wPaper;
    MoveL Offs(pOrigin,40.82,55.88,0.00),v40,z0,tPen\WObj:=wPaper;
    MoveL Offs(pOrigin,41.25,56.95,0.00),v40,z0,tPen\WObj:=wPaper;
    MoveL Offs(pOrigin,24.70,73.50,0.00),v40,z0,tPen\WObj:=wPaper;
    MoveL Offs(pOrigin,25.01,72.47,0.00),v40,z0,tPen\WObj:=wPaper;
    MoveL Offs(pOrigin,42.83,90.28,0.00),v40,z0,tPen\WObj:=wPaper;
    MoveL Offs(pOrigin,43.16,90.89,0.00),v40,z0,tPen\WObj:=wPaper;
    MoveL Offs(pOrigin,57.79,76.25,0.00),v40,z0,tPen\WObj:=wPaper;
    MoveL Offs(pOrigin,58.75,76.78,0.00),v40,z0,tPen\WObj:=wPaper;
    MoveL Offs(pOrigin,68.30,67.24,0.00),v40,z0,tPen\WObj:=wPaper;
    MoveL Offs(pOrigin,68.53,68.19,0.00),v40,z0,tPen\WObj:=wPaper;
    MoveL Offs(pOrigin,86.99,86.65,0.00),v40,z0,tPen\WObj:=wPaper;
    MoveL Offs(pOrigin,87.71,86.65,0.00),v40,z0,tPen\WObj:=wPaper;
    MoveL Offs(pOrigin,58.76,115.61,0.00),v40,z0,tPen\WObj:=wPaper;
    MoveL Offs(pOrigin,59.46,115.87,0.00),v40,z0,tPen\WObj:=wPaper;
    MoveL Offs(pOrigin,72.19,128.60,0.00),v40,z0,tPen\WObj:=wPaper;
    MoveL Offs(pOrigin,71.30,128.70,0.00),v40,z0,tPen\WObj:=wPaper;
    MoveL Offs(pOrigin,60.35,128.70,0.00),v40,z0,tPen\WObj:=wPaper;
    MoveL Offs(pOrigin,60.35,129.75,0.00),v40,z0,tPen\WObj:=wPaper;
    MoveL Offs(pOrigin,71.00,129.75,0.00),v40,z0,tPen\WObj:=wPaper;
    MoveL Offs(pOrigin,71.87,129.77,0.00),v40,z0,tPen\WObj:=wPaper;
    MoveL Offs(pOrigin,59.46,117.36,0.00),v40,z0,tPen\WObj:=wPaper;
    MoveL Offs(pOrigin,60.35,117.08,0.00),v40,z0,tPen\WObj:=wPaper;
    MoveL Offs(pOrigin,75.35,117.08,0.00),v40,z0,tPen\WObj:=wPaper;
    MoveL Offs(pOrigin,76.05,117.53,0.00),v40,z0,tPen\WObj:=wPaper;
    MoveL Offs(pOrigin,59.71,101.19,0.00),v40,z0,tPen\WObj:=wPaper;
    MoveL Offs(pOrigin,60.35,101.24,0.00),v40,z0,tPen\WObj:=wPaper;
    MoveL Offs(pOrigin,81.05,101.24,0.00),v40,z0,tPen\WObj:=wPaper;
    MoveL Offs(pOrigin,81.52,102.09,0.00),v40,z0,tPen\WObj:=wPaper;
    MoveL Offs(pOrigin,72.40,92.97,0.00),v40,fine,tPen\WObj:=wPaper;
    MoveL Offs(pOrigin,72.40,92.97,6.00),v60,z5,tPen\WObj:=wPaper;
    MoveL Offs(pOrigin,73.88,92.96,6.00),vTravel,z5,tPen\WObj:=wPaper;
    MoveL Offs(pOrigin,73.88,92.96,0.00),v60,z0,tPen\WObj:=wPaper;
    MoveL Offs(pOrigin,82.05,101.13,0.00),v40,z0,tPen\WObj:=wPaper;
    MoveL Offs(pOrigin,81.50,100.18,0.00),v40,z0,tPen\WObj:=wPaper;
    MoveL Offs(pOrigin,60.35,100.18,0.00),v40,z0,tPen\WObj:=wPaper;
    MoveL Offs(pOrigin,60.35,99.13,0.00),v40,z0,tPen\WObj:=wPaper;
    MoveL Offs(pOrigin,81.80,99.13,0.00),v40,z0,tPen\WObj:=wPaper;
    MoveL Offs(pOrigin,82.70,98.79,0.00),v40,z0,tPen\WObj:=wPaper;
    MoveL Offs(pOrigin,76.86,92.95,0.00),v40,z0,tPen\WObj:=wPaper;
    MoveL Offs(pOrigin,76.35,92.04,0.00),v40,z0,tPen\WObj:=wPaper;
    MoveL Offs(pOrigin,58.74,109.65,0.00),v40,z0,tPen\WObj:=wPaper;
    MoveL Offs(pOrigin,59.48,109.91,0.00),v40,z0,tPen\WObj:=wPaper;
    MoveL Offs(pOrigin,73.80,124.23,0.00),v40,z0,tPen\WObj:=wPaper;
    MoveL Offs(pOrigin,72.80,124.47,0.00),v40,z0,tPen\WObj:=wPaper;
    MoveL Offs(pOrigin,60.35,124.47,0.00),v40,z0,tPen\WObj:=wPaper;
    MoveL Offs(pOrigin,59.43,124.81,0.00),v40,z0,tPen\WObj:=wPaper;
    MoveL Offs(pOrigin,67.92,133.29,0.00),v40,z0,tPen\WObj:=wPaper;
    MoveL Offs(pOrigin,68.59,134.14,0.00),v40,z0,tPen\WObj:=wPaper;
    MoveL Offs(pOrigin,72.62,130.11,0.00),v40,fine,tPen\WObj:=wPaper;
    MoveL Offs(pOrigin,72.62,130.11,6.00),v60,z5,tPen\WObj:=wPaper;
    MoveL Offs(pOrigin,71.54,130.94,6.00),vTravel,z5,tPen\WObj:=wPaper;
    MoveL Offs(pOrigin,71.54,130.94,0.00),v60,z0,tPen\WObj:=wPaper;
    MoveL Offs(pOrigin,59.45,118.85,0.00),v40,z0,tPen\WObj:=wPaper;
    MoveL Offs(pOrigin,60.35,119.19,0.00),v40,z0,tPen\WObj:=wPaper;
    MoveL Offs(pOrigin,74.60,119.19,0.00),v40,z0,tPen\WObj:=wPaper;
  ENDPROC

  PROC DrawPart5()
    MoveL Offs(pOrigin,75.30,119.76,0.00),v40,z0,tPen\WObj:=wPaper;
    MoveL Offs(pOrigin,59.49,103.96,0.00),v40,z0,tPen\WObj:=wPaper;
    MoveL Offs(pOrigin,58.62,103.80,0.00),v40,z0,tPen\WObj:=wPaper;
    MoveL Offs(pOrigin,70.18,92.24,0.00),v40,z0,tPen\WObj:=wPaper;
    MoveL Offs(pOrigin,70.80,92.86,0.00),v40,z0,tPen\WObj:=wPaper;
    MoveL Offs(pOrigin,81.19,103.26,0.00),v40,z0,tPen\WObj:=wPaper;
    MoveL Offs(pOrigin,80.30,103.35,0.00),v40,z0,tPen\WObj:=wPaper;
    MoveL Offs(pOrigin,60.35,103.35,0.00),v40,z0,tPen\WObj:=wPaper;
    MoveL Offs(pOrigin,60.35,104.41,0.00),v40,z0,tPen\WObj:=wPaper;
    MoveL Offs(pOrigin,80.00,104.41,0.00),v40,z0,tPen\WObj:=wPaper;
    MoveL Offs(pOrigin,80.87,104.43,0.00),v40,z0,tPen\WObj:=wPaper;
    MoveL Offs(pOrigin,69.31,92.87,0.00),v40,z0,tPen\WObj:=wPaper;
    MoveL Offs(pOrigin,68.69,92.24,0.00),v40,z0,tPen\WObj:=wPaper;
    MoveL Offs(pOrigin,58.93,101.99,0.00),v40,z0,tPen\WObj:=wPaper;
    MoveL Offs(pOrigin,59.50,102.47,0.00),v40,z0,tPen\WObj:=wPaper;
    MoveL Offs(pOrigin,75.73,118.70,0.00),v40,z0,tPen\WObj:=wPaper;
    MoveL Offs(pOrigin,76.53,118.74,0.00),v40,z0,tPen\WObj:=wPaper;
    MoveL Offs(pOrigin,61.04,134.23,0.00),v40,fine,tPen\WObj:=wPaper;
    MoveL Offs(pOrigin,61.04,134.23,6.00),v60,z5,tPen\WObj:=wPaper;
    MoveL Offs(pOrigin,60.37,133.21,6.00),vTravel,z5,tPen\WObj:=wPaper;
    MoveL Offs(pOrigin,60.37,133.21,0.00),v60,z0,tPen\WObj:=wPaper;
    MoveL Offs(pOrigin,59.41,132.25,0.00),v40,z0,tPen\WObj:=wPaper;
    MoveL Offs(pOrigin,59.45,132.38,0.00),v40,z0,tPen\WObj:=wPaper;
    MoveL Offs(pOrigin,59.75,133.18,0.00),v40,z0,tPen\WObj:=wPaper;
    MoveL Offs(pOrigin,70.25,133.27,0.00),v40,z0,tPen\WObj:=wPaper;
    MoveL Offs(pOrigin,70.80,132.98,0.00),v40,z0,tPen\WObj:=wPaper;
    MoveL Offs(pOrigin,84.60,92.97,0.00),v40,z0,tPen\WObj:=wPaper;
    MoveL Offs(pOrigin,59.65,92.97,0.00),v40,z0,tPen\WObj:=wPaper;
    MoveL Offs(pOrigin,59.45,132.38,0.00),v40,z0,tPen\WObj:=wPaper;
    MoveL Offs(pOrigin,60.35,131.86,0.00),v40,z0,tPen\WObj:=wPaper;
    MoveL Offs(pOrigin,70.10,131.86,0.00),v40,z0,tPen\WObj:=wPaper;
    MoveL Offs(pOrigin,70.47,132.86,0.00),v40,z0,tPen\WObj:=wPaper;
    MoveL Offs(pOrigin,59.55,121.93,0.00),v40,z0,tPen\WObj:=wPaper;
    MoveL Offs(pOrigin,58.77,121.57,0.00),v40,z0,tPen\WObj:=wPaper;
    MoveL Offs(pOrigin,84.76,95.58,0.00),v40,z0,tPen\WObj:=wPaper;
    MoveL Offs(pOrigin,83.88,95.49,0.00),v40,z0,tPen\WObj:=wPaper;
    MoveL Offs(pOrigin,81.22,92.83,0.00),v40,fine,tPen\WObj:=wPaper;
    MoveL Offs(pOrigin,81.22,92.83,6.00),v60,z5,tPen\WObj:=wPaper;
    MoveL Offs(pOrigin,79.74,92.84,6.00),vTravel,z5,tPen\WObj:=wPaper;
    MoveL Offs(pOrigin,79.74,92.84,0.00),v60,z0,tPen\WObj:=wPaper;
    MoveL Offs(pOrigin,83.34,96.44,0.00),v40,z0,tPen\WObj:=wPaper;
    MoveL Offs(pOrigin,82.85,95.96,0.00),v40,z0,tPen\WObj:=wPaper;
    MoveL Offs(pOrigin,60.35,95.96,0.00),v40,z0,tPen\WObj:=wPaper;
    MoveL Offs(pOrigin,59.73,95.24,0.00),v40,z0,tPen\WObj:=wPaper;
    MoveL Offs(pOrigin,77.76,113.27,0.00),v40,z0,tPen\WObj:=wPaper;
    MoveL Offs(pOrigin,78.53,113.75,0.00),v40,z0,tPen\WObj:=wPaper;
    MoveL Offs(pOrigin,58.81,133.48,0.00),v40,z0,tPen\WObj:=wPaper;
    MoveL Offs(pOrigin,59.77,134.01,0.00),v40,z0,tPen\WObj:=wPaper;
    MoveL Offs(pOrigin,78.11,115.66,0.00),v40,z0,tPen\WObj:=wPaper;
    MoveL Offs(pOrigin,77.01,115.50,0.00),v40,z0,tPen\WObj:=wPaper;
    MoveL Offs(pOrigin,59.51,98.00,0.00),v40,z0,tPen\WObj:=wPaper;
    MoveL Offs(pOrigin,60.20,98.07,0.00),v40,z0,tPen\WObj:=wPaper;
    MoveL Offs(pOrigin,82.10,98.07,0.00),v40,z0,tPen\WObj:=wPaper;
    MoveL Offs(pOrigin,83.13,97.72,0.00),v40,z0,tPen\WObj:=wPaper;
    MoveL Offs(pOrigin,78.35,92.95,0.00),v40,fine,tPen\WObj:=wPaper;
    MoveL Offs(pOrigin,78.35,92.95,6.00),v60,z5,tPen\WObj:=wPaper;
    MoveL Offs(pOrigin,79.00,90.61,6.00),vTravel,z5,tPen\WObj:=wPaper;
    MoveL Offs(pOrigin,79.00,90.61,0.00),v60,z0,tPen\WObj:=wPaper;
    MoveL Offs(pOrigin,59.48,71.09,0.00),v40,z0,tPen\WObj:=wPaper;
    MoveL Offs(pOrigin,58.63,70.93,0.00),v40,z0,tPen\WObj:=wPaper;
    MoveL Offs(pOrigin,62.55,67.01,0.00),v40,fine,tPen\WObj:=wPaper;
    MoveL Offs(pOrigin,62.55,67.01,6.00),v60,z5,tPen\WObj:=wPaper;
    MoveL Offs(pOrigin,62.57,68.21,6.00),vTravel,z5,tPen\WObj:=wPaper;
    MoveL Offs(pOrigin,62.57,68.21,0.00),v60,z0,tPen\WObj:=wPaper;
    MoveL Offs(pOrigin,84.85,90.48,0.00),v40,z0,tPen\WObj:=wPaper;
    MoveL Offs(pOrigin,84.64,91.22,0.00),v40,z0,tPen\WObj:=wPaper;
    MoveL Offs(pOrigin,87.19,88.67,0.00),v40,z0,tPen\WObj:=wPaper;
    MoveL Offs(pOrigin,86.23,88.88,0.00),v40,z0,tPen\WObj:=wPaper;
    MoveL Offs(pOrigin,65.55,68.20,0.00),v40,z0,tPen\WObj:=wPaper;
    MoveL Offs(pOrigin,65.21,67.34,0.00),v40,z0,tPen\WObj:=wPaper;
    MoveL Offs(pOrigin,58.95,73.59,0.00),v40,fine,tPen\WObj:=wPaper;
    MoveL Offs(pOrigin,58.95,73.59,6.00),v60,z5,tPen\WObj:=wPaper;
    MoveL Offs(pOrigin,58.95,72.10,6.00),vTravel,z5,tPen\WObj:=wPaper;
    MoveL Offs(pOrigin,58.95,72.10,0.00),v60,z0,tPen\WObj:=wPaper;
    MoveL Offs(pOrigin,64.04,67.01,0.00),v40,z0,tPen\WObj:=wPaper;
    MoveL Offs(pOrigin,64.06,68.21,0.00),v40,z0,tPen\WObj:=wPaper;
    MoveL Offs(pOrigin,85.81,89.95,0.00),v40,fine,tPen\WObj:=wPaper;
    MoveL Offs(pOrigin,85.81,89.95,6.00),v60,z5,tPen\WObj:=wPaper;
    MoveL Offs(pOrigin,84.50,89.62,6.00),vTravel,z5,tPen\WObj:=wPaper;
    MoveL Offs(pOrigin,84.50,89.62,0.00),v60,z0,tPen\WObj:=wPaper;
    MoveL Offs(pOrigin,63.95,89.62,0.00),v40,z0,tPen\WObj:=wPaper;
    MoveL Offs(pOrigin,63.89,90.44,0.00),v40,z0,tPen\WObj:=wPaper;
    MoveL Offs(pOrigin,59.86,86.41,0.00),v40,z0,tPen\WObj:=wPaper;
    MoveL Offs(pOrigin,60.65,86.46,0.00),v40,z0,tPen\WObj:=wPaper;
    MoveL Offs(pOrigin,86.15,86.46,0.00),v40,z0,tPen\WObj:=wPaper;
    MoveL Offs(pOrigin,86.45,85.40,0.00),v40,z0,tPen\WObj:=wPaper;
    MoveL Offs(pOrigin,60.65,85.40,0.00),v40,z0,tPen\WObj:=wPaper;
    MoveL Offs(pOrigin,60.50,84.34,0.00),v40,z0,tPen\WObj:=wPaper;
    MoveL Offs(pOrigin,86.90,84.34,0.00),v40,z0,tPen\WObj:=wPaper;
    MoveL Offs(pOrigin,87.74,84.41,0.00),v40,z0,tPen\WObj:=wPaper;
    MoveL Offs(pOrigin,71.51,68.18,0.00),v40,z0,tPen\WObj:=wPaper;
    MoveL Offs(pOrigin,71.28,67.25,0.00),v40,z0,tPen\WObj:=wPaper;
    MoveL Offs(pOrigin,59.08,79.44,0.00),v40,z0,tPen\WObj:=wPaper;
    MoveL Offs(pOrigin,59.67,78.75,0.00),v40,z0,tPen\WObj:=wPaper;
    MoveL Offs(pOrigin,71.45,90.52,0.00),v40,z0,tPen\WObj:=wPaper;
    MoveL Offs(pOrigin,71.34,91.07,0.00),v40,z0,tPen\WObj:=wPaper;
    MoveL Offs(pOrigin,94.68,67.74,0.00),v40,fine,tPen\WObj:=wPaper;
    MoveL Offs(pOrigin,94.68,67.74,6.00),v60,z5,tPen\WObj:=wPaper;
    MoveL Offs(pOrigin,93.96,66.74,6.00),vTravel,z5,tPen\WObj:=wPaper;
    MoveL Offs(pOrigin,93.96,66.74,0.00),v60,z0,tPen\WObj:=wPaper;
    MoveL Offs(pOrigin,78.68,51.46,0.00),v40,fine,tPen\WObj:=wPaper;
    MoveL Offs(pOrigin,78.68,51.46,6.00),v60,z5,tPen\WObj:=wPaper;
    MoveL Offs(pOrigin,78.80,53.72,6.00),vTravel,z5,tPen\WObj:=wPaper;
    MoveL Offs(pOrigin,78.80,53.72,0.00),v60,z0,tPen\WObj:=wPaper;
    MoveL Offs(pOrigin,97.85,53.72,0.00),v40,z0,tPen\WObj:=wPaper;
    MoveL Offs(pOrigin,98.78,53.64,0.00),v40,z0,tPen\WObj:=wPaper;
    MoveL Offs(pOrigin,95.81,50.67,0.00),v40,z0,tPen\WObj:=wPaper;
    MoveL Offs(pOrigin,96.33,49.66,0.00),v40,z0,tPen\WObj:=wPaper;
    MoveL Offs(pOrigin,59.10,86.89,0.00),v40,z0,tPen\WObj:=wPaper;
    MoveL Offs(pOrigin,59.75,87.79,0.00),v40,z0,tPen\WObj:=wPaper;
    MoveL Offs(pOrigin,62.19,90.23,0.00),v40,z0,tPen\WObj:=wPaper;
    MoveL Offs(pOrigin,62.51,90.94,0.00),v40,z0,tPen\WObj:=wPaper;
    MoveL Offs(pOrigin,99.85,53.61,0.00),v40,fine,tPen\WObj:=wPaper;
    MoveL Offs(pOrigin,99.85,53.61,6.00),v60,z5,tPen\WObj:=wPaper;
    MoveL Offs(pOrigin,99.21,52.58,6.00),vTravel,z5,tPen\WObj:=wPaper;
    MoveL Offs(pOrigin,99.21,52.58,0.00),v60,z0,tPen\WObj:=wPaper;
    MoveL Offs(pOrigin,97.30,50.67,0.00),v40,z0,tPen\WObj:=wPaper;
    MoveL Offs(pOrigin,97.71,49.77,0.00),v40,z0,tPen\WObj:=wPaper;
    MoveL Offs(pOrigin,59.10,88.38,0.00),v40,fine,tPen\WObj:=wPaper;
    MoveL Offs(pOrigin,59.10,88.38,6.00),v60,z5,tPen\WObj:=wPaper;
  ENDPROC

  PROC DrawPart6()
    MoveL Offs(pOrigin,59.85,89.38,6.00),vTravel,z5,tPen\WObj:=wPaper;
    MoveL Offs(pOrigin,59.85,89.38,0.00),v60,z0,tPen\WObj:=wPaper;
    MoveL Offs(pOrigin,60.70,90.23,0.00),v40,z0,tPen\WObj:=wPaper;
    MoveL Offs(pOrigin,61.03,90.94,0.00),v40,z0,tPen\WObj:=wPaper;
    MoveL Offs(pOrigin,100.06,51.91,0.00),v40,fine,tPen\WObj:=wPaper;
    MoveL Offs(pOrigin,100.06,51.91,6.00),v60,z5,tPen\WObj:=wPaper;
    MoveL Offs(pOrigin,99.95,50.52,6.00),vTravel,z5,tPen\WObj:=wPaper;
    MoveL Offs(pOrigin,99.95,50.52,0.00),v60,z0,tPen\WObj:=wPaper;
    MoveL Offs(pOrigin,59.75,90.72,0.00),v40,z0,tPen\WObj:=wPaper;
    MoveL Offs(pOrigin,59.11,89.87,0.00),v40,z0,tPen\WObj:=wPaper;
    MoveL Offs(pOrigin,98.99,49.99,0.00),v40,fine,tPen\WObj:=wPaper;
    MoveL Offs(pOrigin,98.99,49.99,6.00),v60,z5,tPen\WObj:=wPaper;
    MoveL Offs(pOrigin,95.16,49.34,6.00),vTravel,z5,tPen\WObj:=wPaper;
    MoveL Offs(pOrigin,95.16,49.34,0.00),v60,z0,tPen\WObj:=wPaper;
    MoveL Offs(pOrigin,59.09,85.40,0.00),v40,fine,tPen\WObj:=wPaper;
    MoveL Offs(pOrigin,59.09,85.40,6.00),v60,z5,tPen\WObj:=wPaper;
    MoveL Offs(pOrigin,60.65,87.51,6.00),vTravel,z5,tPen\WObj:=wPaper;
    MoveL Offs(pOrigin,60.65,87.51,0.00),v60,z0,tPen\WObj:=wPaper;
    MoveL Offs(pOrigin,85.70,87.51,0.00),v40,z0,tPen\WObj:=wPaper;
    MoveL Offs(pOrigin,86.56,87.71,0.00),v40,z0,tPen\WObj:=wPaper;
    MoveL Offs(pOrigin,67.04,68.20,0.00),v40,z0,tPen\WObj:=wPaper;
    MoveL Offs(pOrigin,66.70,67.34,0.00),v40,z0,tPen\WObj:=wPaper;
    MoveL Offs(pOrigin,58.75,75.30,0.00),v40,fine,tPen\WObj:=wPaper;
    MoveL Offs(pOrigin,58.75,75.30,6.00),v60,z5,tPen\WObj:=wPaper;
    MoveL Offs(pOrigin,60.50,73.78,6.00),vTravel,z5,tPen\WObj:=wPaper;
    MoveL Offs(pOrigin,60.50,73.78,0.00),v60,z0,tPen\WObj:=wPaper;
    MoveL Offs(pOrigin,90.50,73.78,0.00),v40,fine,tPen\WObj:=wPaper;
    MoveL Offs(pOrigin,90.50,73.78,6.00),v60,z5,tPen\WObj:=wPaper;
    MoveL Offs(pOrigin,90.85,75.58,6.00),vTravel,z5,tPen\WObj:=wPaper;
    MoveL Offs(pOrigin,90.85,75.58,0.00),v60,z0,tPen\WObj:=wPaper;
    MoveL Offs(pOrigin,75.68,60.41,0.00),v40,z0,tPen\WObj:=wPaper;
    MoveL Offs(pOrigin,76.25,61.11,0.00),v40,z0,tPen\WObj:=wPaper;
    MoveL Offs(pOrigin,95.15,61.11,0.00),v40,z0,tPen\WObj:=wPaper;
    MoveL Offs(pOrigin,95.99,61.31,0.00),v40,z0,tPen\WObj:=wPaper;
    MoveL Offs(pOrigin,85.39,50.70,0.00),v40,fine,tPen\WObj:=wPaper;
    MoveL Offs(pOrigin,85.39,50.70,6.00),v60,z5,tPen\WObj:=wPaper;
    MoveL Offs(pOrigin,87.71,49.32,6.00),vTravel,z5,tPen\WObj:=wPaper;
    MoveL Offs(pOrigin,87.71,49.32,0.00),v60,z0,tPen\WObj:=wPaper;
    MoveL Offs(pOrigin,73.39,63.64,0.00),v40,fine,tPen\WObj:=wPaper;
    MoveL Offs(pOrigin,73.39,63.64,6.00),v60,z5,tPen\WObj:=wPaper;
    MoveL Offs(pOrigin,74.61,63.81,6.00),vTravel,z5,tPen\WObj:=wPaper;
    MoveL Offs(pOrigin,74.61,63.81,0.00),v60,z0,tPen\WObj:=wPaper;
    MoveL Offs(pOrigin,89.77,78.98,0.00),v40,z0,tPen\WObj:=wPaper;
    MoveL Offs(pOrigin,90.77,79.11,0.00),v40,z0,tPen\WObj:=wPaper;
    MoveL Offs(pOrigin,43.26,126.63,0.00),v40,fine,tPen\WObj:=wPaper;
    MoveL Offs(pOrigin,43.26,126.63,6.00),v60,z5,tPen\WObj:=wPaper;
    MoveL Offs(pOrigin,43.58,127.80,6.00),vTravel,z5,tPen\WObj:=wPaper;
    MoveL Offs(pOrigin,43.58,127.80,0.00),v60,z0,tPen\WObj:=wPaper;
    MoveL Offs(pOrigin,89.72,81.66,0.00),v40,z0,tPen\WObj:=wPaper;
    MoveL Offs(pOrigin,88.92,81.11,0.00),v40,z0,tPen\WObj:=wPaper;
    MoveL Offs(pOrigin,73.85,66.05,0.00),v40,z0,tPen\WObj:=wPaper;
    MoveL Offs(pOrigin,74.60,66.39,0.00),v40,z0,tPen\WObj:=wPaper;
    MoveL Offs(pOrigin,93.20,66.39,0.00),v40,z0,tPen\WObj:=wPaper;
    MoveL Offs(pOrigin,93.65,65.34,0.00),v40,z0,tPen\WObj:=wPaper;
    MoveL Offs(pOrigin,74.90,65.34,0.00),v40,z0,tPen\WObj:=wPaper;
    MoveL Offs(pOrigin,74.28,64.99,0.00),v40,z0,tPen\WObj:=wPaper;
    MoveL Offs(pOrigin,89.34,80.05,0.00),v40,z0,tPen\WObj:=wPaper;
    MoveL Offs(pOrigin,88.25,80.12,0.00),v40,z0,tPen\WObj:=wPaper;
    MoveL Offs(pOrigin,60.65,80.12,0.00),v40,z0,tPen\WObj:=wPaper;
    MoveL Offs(pOrigin,60.65,79.06,0.00),v40,z0,tPen\WObj:=wPaper;
    MoveL Offs(pOrigin,88.70,79.06,0.00),v40,z0,tPen\WObj:=wPaper;
    MoveL Offs(pOrigin,89.00,78.01,0.00),v40,z0,tPen\WObj:=wPaper;
    MoveL Offs(pOrigin,60.65,78.01,0.00),v40,fine,tPen\WObj:=wPaper;
    MoveL Offs(pOrigin,60.65,78.01,6.00),v60,z5,tPen\WObj:=wPaper;
    MoveL Offs(pOrigin,58.97,78.06,6.00),vTravel,z5,tPen\WObj:=wPaper;
    MoveL Offs(pOrigin,58.97,78.06,0.00),v60,z0,tPen\WObj:=wPaper;
    MoveL Offs(pOrigin,70.00,67.03,0.00),v40,z0,tPen\WObj:=wPaper;
    MoveL Offs(pOrigin,70.02,68.19,0.00),v40,z0,tPen\WObj:=wPaper;
    MoveL Offs(pOrigin,87.31,85.48,0.00),v40,fine,tPen\WObj:=wPaper;
    MoveL Offs(pOrigin,87.31,85.48,6.00),v60,z5,tPen\WObj:=wPaper;
    MoveL Offs(pOrigin,88.98,83.89,6.00),vTravel,z5,tPen\WObj:=wPaper;
    MoveL Offs(pOrigin,88.98,83.89,0.00),v60,z0,tPen\WObj:=wPaper;
    MoveL Offs(pOrigin,58.75,114.12,0.00),v40,z0,tPen\WObj:=wPaper;
    MoveL Offs(pOrigin,59.46,114.38,0.00),v40,z0,tPen\WObj:=wPaper;
    MoveL Offs(pOrigin,72.62,127.53,0.00),v40,z0,tPen\WObj:=wPaper;
    MoveL Offs(pOrigin,73.36,127.88,0.00),v40,z0,tPen\WObj:=wPaper;
    MoveL Offs(pOrigin,67.10,134.14,0.00),v40,z0,tPen\WObj:=wPaper;
    MoveL Offs(pOrigin,66.43,133.30,0.00),v40,z0,tPen\WObj:=wPaper;
    MoveL Offs(pOrigin,59.43,126.30,0.00),v40,z0,tPen\WObj:=wPaper;
    MoveL Offs(pOrigin,60.35,126.58,0.00),v40,z0,tPen\WObj:=wPaper;
    MoveL Offs(pOrigin,72.05,126.58,0.00),v40,z0,tPen\WObj:=wPaper;
    MoveL Offs(pOrigin,73.04,126.47,0.00),v40,z0,tPen\WObj:=wPaper;
    MoveL Offs(pOrigin,59.47,112.89,0.00),v40,z0,tPen\WObj:=wPaper;
    MoveL Offs(pOrigin,60.35,112.86,0.00),v40,z0,tPen\WObj:=wPaper;
    MoveL Offs(pOrigin,76.85,112.86,0.00),v40,z0,tPen\WObj:=wPaper;
    MoveL Offs(pOrigin,77.15,111.80,0.00),v40,z0,tPen\WObj:=wPaper;
    MoveL Offs(pOrigin,60.35,111.80,0.00),v40,z0,tPen\WObj:=wPaper;
    MoveL Offs(pOrigin,59.47,111.40,0.00),v40,z0,tPen\WObj:=wPaper;
    MoveL Offs(pOrigin,73.47,125.40,0.00),v40,z0,tPen\WObj:=wPaper;
    MoveL Offs(pOrigin,74.53,125.23,0.00),v40,z0,tPen\WObj:=wPaper;
    MoveL Offs(pOrigin,65.62,134.14,0.00),v40,z0,tPen\WObj:=wPaper;
    MoveL Offs(pOrigin,64.94,133.30,0.00),v40,z0,tPen\WObj:=wPaper;
    MoveL Offs(pOrigin,59.43,127.78,0.00),v40,z0,tPen\WObj:=wPaper;
    MoveL Offs(pOrigin,60.35,127.64,0.00),v40,z0,tPen\WObj:=wPaper;
    MoveL Offs(pOrigin,71.75,127.64,0.00),v40,fine,tPen\WObj:=wPaper;
    MoveL Offs(pOrigin,71.75,127.64,6.00),v60,z5,tPen\WObj:=wPaper;
    MoveL Offs(pOrigin,72.35,125.53,6.00),vTravel,z5,tPen\WObj:=wPaper;
    MoveL Offs(pOrigin,72.35,125.53,0.00),v60,z0,tPen\WObj:=wPaper;
    MoveL Offs(pOrigin,60.35,125.53,0.00),v40,fine,tPen\WObj:=wPaper;
    MoveL Offs(pOrigin,60.35,125.53,6.00),v60,z5,tPen\WObj:=wPaper;
    MoveL Offs(pOrigin,60.35,123.42,6.00),vTravel,z5,tPen\WObj:=wPaper;
    MoveL Offs(pOrigin,60.35,123.42,0.00),v60,z0,tPen\WObj:=wPaper;
    MoveL Offs(pOrigin,73.10,123.42,0.00),v40,z0,tPen\WObj:=wPaper;
    MoveL Offs(pOrigin,73.55,122.36,0.00),v40,z0,tPen\WObj:=wPaper;
    MoveL Offs(pOrigin,60.35,122.36,0.00),v40,z0,tPen\WObj:=wPaper;
    MoveL Offs(pOrigin,60.35,121.30,0.00),v40,z0,tPen\WObj:=wPaper;
    MoveL Offs(pOrigin,73.85,121.30,0.00),v40,z0,tPen\WObj:=wPaper;
    MoveL Offs(pOrigin,74.55,122.00,0.00),v40,z0,tPen\WObj:=wPaper;
    MoveL Offs(pOrigin,59.49,106.94,0.00),v40,z0,tPen\WObj:=wPaper;
    MoveL Offs(pOrigin,58.73,106.67,0.00),v40,z0,tPen\WObj:=wPaper;
    MoveL Offs(pOrigin,92.88,72.52,0.00),v40,fine,tPen\WObj:=wPaper;
    MoveL Offs(pOrigin,92.88,72.52,6.00),v60,z5,tPen\WObj:=wPaper;
    MoveL Offs(pOrigin,94.36,69.55,6.00),vTravel,z5,tPen\WObj:=wPaper;
    MoveL Offs(pOrigin,94.36,69.55,0.00),v60,z0,tPen\WObj:=wPaper;
    MoveL Offs(pOrigin,58.62,105.29,0.00),v40,z0,tPen\WObj:=wPaper;
    MoveL Offs(pOrigin,59.49,105.45,0.00),v40,z0,tPen\WObj:=wPaper;
    MoveL Offs(pOrigin,74.98,120.93,0.00),v40,z0,tPen\WObj:=wPaper;
    MoveL Offs(pOrigin,74.30,120.25,0.00),v40,z0,tPen\WObj:=wPaper;
    MoveL Offs(pOrigin,60.35,120.25,0.00),v40,z0,tPen\WObj:=wPaper;
    MoveL Offs(pOrigin,59.55,120.45,0.00),v40,z0,tPen\WObj:=wPaper;
  ENDPROC

  PROC DrawPart7()
    MoveL Offs(pOrigin,71.22,132.11,0.00),v40,z0,tPen\WObj:=wPaper;
    MoveL Offs(pOrigin,72.31,131.92,0.00),v40,z0,tPen\WObj:=wPaper;
    MoveL Offs(pOrigin,70.40,133.83,0.00),v40,fine,tPen\WObj:=wPaper;
    MoveL Offs(pOrigin,70.40,133.83,6.00),v60,z5,tPen\WObj:=wPaper;
    MoveL Offs(pOrigin,69.30,133.18,6.00),vTravel,z5,tPen\WObj:=wPaper;
    MoveL Offs(pOrigin,69.30,133.18,0.00),v60,z0,tPen\WObj:=wPaper;
    MoveL Offs(pOrigin,59.54,123.42,0.00),v40,fine,tPen\WObj:=wPaper;
    MoveL Offs(pOrigin,59.54,123.42,6.00),v60,z5,tPen\WObj:=wPaper;
    MoveL Offs(pOrigin,57.92,122.41,6.00),vTravel,z5,tPen\WObj:=wPaper;
    MoveL Offs(pOrigin,57.92,122.41,0.00),v60,z0,tPen\WObj:=wPaper;
    MoveL Offs(pOrigin,46.47,133.87,0.00),v40,z0,tPen\WObj:=wPaper;
    MoveL Offs(pOrigin,46.45,133.07,0.00),v40,z0,tPen\WObj:=wPaper;
    MoveL Offs(pOrigin,57.15,133.07,0.00),v40,z0,tPen\WObj:=wPaper;
    MoveL Offs(pOrigin,57.15,92.97,0.00),v40,z0,tPen\WObj:=wPaper;
    MoveL Offs(pOrigin,32.65,92.97,0.00),v40,z0,tPen\WObj:=wPaper;
    MoveL Offs(pOrigin,33.15,95.18,0.00),v40,z0,tPen\WObj:=wPaper;
    MoveL Offs(pOrigin,46.45,133.07,0.00),v40,z0,tPen\WObj:=wPaper;
    MoveL Offs(pOrigin,46.97,133.25,0.00),v40,z0,tPen\WObj:=wPaper;
    MoveL Offs(pOrigin,45.90,132.18,0.00),v40,z0,tPen\WObj:=wPaper;
    MoveL Offs(pOrigin,46.85,131.86,0.00),v40,z0,tPen\WObj:=wPaper;
    MoveL Offs(pOrigin,56.30,131.86,0.00),v40,z0,tPen\WObj:=wPaper;
    MoveL Offs(pOrigin,57.18,131.51,0.00),v40,z0,tPen\WObj:=wPaper;
    MoveL Offs(pOrigin,39.89,114.23,0.00),v40,z0,tPen\WObj:=wPaper;
    MoveL Offs(pOrigin,39.18,114.28,0.00),v40,z0,tPen\WObj:=wPaper;
    MoveL Offs(pOrigin,57.64,95.82,0.00),v40,z0,tPen\WObj:=wPaper;
    MoveL Offs(pOrigin,56.86,95.35,0.00),v40,z0,tPen\WObj:=wPaper;
    MoveL Offs(pOrigin,54.63,93.12,0.00),v40,z0,tPen\WObj:=wPaper;
    MoveL Offs(pOrigin,55.07,92.41,0.00),v40,z0,tPen\WObj:=wPaper;
    MoveL Offs(pOrigin,37.57,109.91,0.00),v40,z0,tPen\WObj:=wPaper;
    MoveL Offs(pOrigin,38.20,109.55,0.00),v40,z0,tPen\WObj:=wPaper;
    MoveL Offs(pOrigin,57.19,128.54,0.00),v40,z0,tPen\WObj:=wPaper;
    MoveL Offs(pOrigin,56.45,128.70,0.00),v40,z0,tPen\WObj:=wPaper;
    MoveL Offs(pOrigin,45.80,128.70,0.00),v40,z0,tPen\WObj:=wPaper;
    MoveL Offs(pOrigin,46.10,129.75,0.00),v40,z0,tPen\WObj:=wPaper;
    MoveL Offs(pOrigin,56.45,129.75,0.00),v40,z0,tPen\WObj:=wPaper;
    MoveL Offs(pOrigin,57.19,130.03,0.00),v40,z0,tPen\WObj:=wPaper;
    MoveL Offs(pOrigin,38.94,111.78,0.00),v40,z0,tPen\WObj:=wPaper;
    MoveL Offs(pOrigin,38.22,112.25,0.00),v40,z0,tPen\WObj:=wPaper;
    MoveL Offs(pOrigin,57.31,93.16,0.00),v40,z0,tPen\WObj:=wPaper;
    MoveL Offs(pOrigin,56.86,93.86,0.00),v40,z0,tPen\WObj:=wPaper;
    MoveL Offs(pOrigin,56.23,93.22,0.00),v40,z0,tPen\WObj:=wPaper;
    MoveL Offs(pOrigin,56.35,92.63,0.00),v40,z0,tPen\WObj:=wPaper;
    MoveL Offs(pOrigin,37.79,111.19,0.00),v40,fine,tPen\WObj:=wPaper;
    MoveL Offs(pOrigin,37.79,111.19,6.00),v60,z5,tPen\WObj:=wPaper;
    MoveL Offs(pOrigin,39.50,110.74,6.00),vTravel,z5,tPen\WObj:=wPaper;
    MoveL Offs(pOrigin,39.50,110.74,0.00),v60,z0,tPen\WObj:=wPaper;
    MoveL Offs(pOrigin,56.30,110.74,0.00),v40,z0,tPen\WObj:=wPaper;
    MoveL Offs(pOrigin,57.03,110.45,0.00),v40,z0,tPen\WObj:=wPaper;
    MoveL Offs(pOrigin,39.74,93.17,0.00),v40,z0,tPen\WObj:=wPaper;
    MoveL Offs(pOrigin,40.29,92.26,0.00),v40,z0,tPen\WObj:=wPaper;
    MoveL Offs(pOrigin,33.71,98.84,0.00),v40,z0,tPen\WObj:=wPaper;
    MoveL Offs(pOrigin,34.19,98.07,0.00),v40,z0,tPen\WObj:=wPaper;
    MoveL Offs(pOrigin,57.21,121.09,0.00),v40,z0,tPen\WObj:=wPaper;
    MoveL Offs(pOrigin,56.30,121.30,0.00),v40,z0,tPen\WObj:=wPaper;
    MoveL Offs(pOrigin,43.25,121.30,0.00),v40,z0,tPen\WObj:=wPaper;
    MoveL Offs(pOrigin,43.55,122.36,0.00),v40,z0,tPen\WObj:=wPaper;
    MoveL Offs(pOrigin,56.30,122.36,0.00),v40,z0,tPen\WObj:=wPaper;
    MoveL Offs(pOrigin,57.21,122.58,0.00),v40,z0,tPen\WObj:=wPaper;
    MoveL Offs(pOrigin,34.93,100.31,0.00),v40,z0,tPen\WObj:=wPaper;
    MoveL Offs(pOrigin,35.75,100.18,0.00),v40,z0,tPen\WObj:=wPaper;
    MoveL Offs(pOrigin,56.45,100.18,0.00),v40,z0,tPen\WObj:=wPaper;
    MoveL Offs(pOrigin,57.06,100.03,0.00),v40,z0,tPen\WObj:=wPaper;
    MoveL Offs(pOrigin,50.27,93.24,0.00),v40,z0,tPen\WObj:=wPaper;
    MoveL Offs(pOrigin,50.61,92.40,0.00),v40,z0,tPen\WObj:=wPaper;
    MoveL Offs(pOrigin,36.39,106.61,0.00),v40,z0,tPen\WObj:=wPaper;
    MoveL Offs(pOrigin,36.93,107.57,0.00),v40,z0,tPen\WObj:=wPaper;
    MoveL Offs(pOrigin,52.09,92.40,0.00),v40,z0,tPen\WObj:=wPaper;
    MoveL Offs(pOrigin,51.76,93.24,0.00),v40,z0,tPen\WObj:=wPaper;
    MoveL Offs(pOrigin,57.06,98.54,0.00),v40,z0,tPen\WObj:=wPaper;
    MoveL Offs(pOrigin,57.86,98.59,0.00),v40,z0,tPen\WObj:=wPaper;
    MoveL Offs(pOrigin,39.93,116.51,0.00),v40,z0,tPen\WObj:=wPaper;
    MoveL Offs(pOrigin,40.63,116.46,0.00),v40,z0,tPen\WObj:=wPaper;
    MoveL Offs(pOrigin,56.86,132.69,0.00),v40,z0,tPen\WObj:=wPaper;
    MoveL Offs(pOrigin,57.11,133.69,0.00),v40,z0,tPen\WObj:=wPaper;
    MoveL Offs(pOrigin,79.91,110.88,0.00),v40,fine,tPen\WObj:=wPaper;
    MoveL Offs(pOrigin,79.91,110.88,6.00),v60,z5,tPen\WObj:=wPaper;
    MoveL Offs(pOrigin,78.51,111.03,6.00),vTravel,z5,tPen\WObj:=wPaper;
    MoveL Offs(pOrigin,78.51,111.03,0.00),v60,z0,tPen\WObj:=wPaper;
    MoveL Offs(pOrigin,60.59,93.11,0.00),v40,z0,tPen\WObj:=wPaper;
    MoveL Offs(pOrigin,60.65,93.85,0.00),v40,z0,tPen\WObj:=wPaper;
    MoveL Offs(pOrigin,83.30,93.85,0.00),v40,z0,tPen\WObj:=wPaper;
    MoveL Offs(pOrigin,82.82,92.94,0.00),v40,z0,tPen\WObj:=wPaper;
    MoveL Offs(pOrigin,84.30,94.42,0.00),v40,z0,tPen\WObj:=wPaper;
    MoveL Offs(pOrigin,83.30,94.90,0.00),v40,z0,tPen\WObj:=wPaper;
    MoveL Offs(pOrigin,60.35,94.90,0.00),v40,z0,tPen\WObj:=wPaper;
    MoveL Offs(pOrigin,59.84,93.85,0.00),v40,z0,tPen\WObj:=wPaper;
    MoveL Offs(pOrigin,78.08,112.10,0.00),v40,fine,tPen\WObj:=wPaper;
    MoveL Offs(pOrigin,78.08,112.10,6.00),v60,z5,tPen\WObj:=wPaper;
    MoveL Offs(pOrigin,77.60,110.74,6.00),vTravel,z5,tPen\WObj:=wPaper;
    MoveL Offs(pOrigin,77.60,110.74,0.00),v60,z0,tPen\WObj:=wPaper;
    MoveL Offs(pOrigin,60.35,110.74,0.00),v40,z0,tPen\WObj:=wPaper;
    MoveL Offs(pOrigin,60.35,109.69,0.00),v40,z0,tPen\WObj:=wPaper;
    MoveL Offs(pOrigin,78.05,109.69,0.00),v40,z0,tPen\WObj:=wPaper;
    MoveL Offs(pOrigin,78.84,109.86,0.00),v40,z0,tPen\WObj:=wPaper;
    MoveL Offs(pOrigin,62.08,93.10,0.00),v40,z0,tPen\WObj:=wPaper;
    MoveL Offs(pOrigin,62.52,92.43,0.00),v40,z0,tPen\WObj:=wPaper;
    MoveL Offs(pOrigin,59.02,95.93,0.00),v40,z0,tPen\WObj:=wPaper;
    MoveL Offs(pOrigin,59.51,96.51,0.00),v40,z0,tPen\WObj:=wPaper;
    MoveL Offs(pOrigin,77.23,114.23,0.00),v40,z0,tPen\WObj:=wPaper;
    MoveL Offs(pOrigin,76.55,113.91,0.00),v40,z0,tPen\WObj:=wPaper;
    MoveL Offs(pOrigin,60.35,113.91,0.00),v40,z0,tPen\WObj:=wPaper;
    MoveL Offs(pOrigin,60.35,114.97,0.00),v40,z0,tPen\WObj:=wPaper;
    MoveL Offs(pOrigin,76.25,114.97,0.00),v40,z0,tPen\WObj:=wPaper;
    MoveL Offs(pOrigin,75.80,116.02,0.00),v40,z0,tPen\WObj:=wPaper;
    MoveL Offs(pOrigin,60.35,116.02,0.00),v40,fine,tPen\WObj:=wPaper;
    MoveL Offs(pOrigin,60.35,116.02,6.00),v60,z5,tPen\WObj:=wPaper;
    MoveL Offs(pOrigin,60.35,118.14,6.00),vTravel,z5,tPen\WObj:=wPaper;
    MoveL Offs(pOrigin,60.35,118.14,0.00),v60,z0,tPen\WObj:=wPaper;
    MoveL Offs(pOrigin,74.90,118.14,0.00),v40,fine,tPen\WObj:=wPaper;
    MoveL Offs(pOrigin,74.90,118.14,6.00),v60,z5,tPen\WObj:=wPaper;
    MoveL Offs(pOrigin,76.48,116.46,6.00),vTravel,z5,tPen\WObj:=wPaper;
    MoveL Offs(pOrigin,76.48,116.46,0.00),v60,z0,tPen\WObj:=wPaper;
    MoveL Offs(pOrigin,59.51,99.49,0.00),v40,z0,tPen\WObj:=wPaper;
    MoveL Offs(pOrigin,59.03,98.91,0.00),v40,z0,tPen\WObj:=wPaper;
    MoveL Offs(pOrigin,65.82,92.12,0.00),v40,z0,tPen\WObj:=wPaper;
    MoveL Offs(pOrigin,66.44,92.98,0.00),v40,z0,tPen\WObj:=wPaper;
    MoveL Offs(pOrigin,80.02,106.56,0.00),v40,z0,tPen\WObj:=wPaper;
    MoveL Offs(pOrigin,80.75,107.06,0.00),v40,z0,tPen\WObj:=wPaper;
    MoveL Offs(pOrigin,53.60,134.21,0.00),v40,z0,tPen\WObj:=wPaper;
    MoveL Offs(pOrigin,53.03,133.33,0.00),v40,z0,tPen\WObj:=wPaper;
  ENDPROC

  PROC DrawPart8()
    MoveL Offs(pOrigin,42.74,123.05,0.00),v40,z0,tPen\WObj:=wPaper;
    MoveL Offs(pOrigin,42.08,123.33,0.00),v40,z0,tPen\WObj:=wPaper;
    MoveL Offs(pOrigin,57.78,107.63,0.00),v40,z0,tPen\WObj:=wPaper;
    MoveL Offs(pOrigin,57.04,107.48,0.00),v40,z0,tPen\WObj:=wPaper;
    MoveL Offs(pOrigin,42.72,93.16,0.00),v40,z0,tPen\WObj:=wPaper;
    MoveL Offs(pOrigin,43.16,92.38,0.00),v40,z0,tPen\WObj:=wPaper;
    MoveL Offs(pOrigin,34.36,101.18,0.00),v40,z0,tPen\WObj:=wPaper;
    MoveL Offs(pOrigin,34.89,102.14,0.00),v40,z0,tPen\WObj:=wPaper;
    MoveL Offs(pOrigin,44.75,92.27,0.00),v40,z0,tPen\WObj:=wPaper;
    MoveL Offs(pOrigin,44.21,93.15,0.00),v40,z0,tPen\WObj:=wPaper;
    MoveL Offs(pOrigin,57.04,105.99,0.00),v40,z0,tPen\WObj:=wPaper;
    MoveL Offs(pOrigin,57.77,106.14,0.00),v40,z0,tPen\WObj:=wPaper;
    MoveL Offs(pOrigin,41.54,122.37,0.00),v40,fine,tPen\WObj:=wPaper;
    MoveL Offs(pOrigin,41.54,122.37,6.00),v60,z5,tPen\WObj:=wPaper;
    MoveL Offs(pOrigin,41.22,121.20,6.00),vTravel,z5,tPen\WObj:=wPaper;
    MoveL Offs(pOrigin,41.22,121.20,0.00),v60,z0,tPen\WObj:=wPaper;
    MoveL Offs(pOrigin,57.87,104.54,0.00),v40,z0,tPen\WObj:=wPaper;
    MoveL Offs(pOrigin,57.05,104.50,0.00),v40,z0,tPen\WObj:=wPaper;
    MoveL Offs(pOrigin,45.70,93.15,0.00),v40,z0,tPen\WObj:=wPaper;
    MoveL Offs(pOrigin,46.14,92.38,0.00),v40,z0,tPen\WObj:=wPaper;
    MoveL Offs(pOrigin,35.43,103.10,0.00),v40,z0,tPen\WObj:=wPaper;
    MoveL Offs(pOrigin,35.67,102.54,0.00),v40,z0,tPen\WObj:=wPaper;
    MoveL Offs(pOrigin,57.20,124.07,0.00),v40,z0,tPen\WObj:=wPaper;
    MoveL Offs(pOrigin,56.30,124.47,0.00),v40,z0,tPen\WObj:=wPaper;
    MoveL Offs(pOrigin,44.45,124.47,0.00),v40,z0,tPen\WObj:=wPaper;
    MoveL Offs(pOrigin,44.75,125.53,0.00),v40,z0,tPen\WObj:=wPaper;
    MoveL Offs(pOrigin,56.30,125.53,0.00),v40,z0,tPen\WObj:=wPaper;
    MoveL Offs(pOrigin,57.20,125.56,0.00),v40,z0,tPen\WObj:=wPaper;
    MoveL Offs(pOrigin,36.73,105.09,0.00),v40,z0,tPen\WObj:=wPaper;
    MoveL Offs(pOrigin,36.18,105.33,0.00),v40,z0,tPen\WObj:=wPaper;
    MoveL Offs(pOrigin,48.90,92.60,0.00),v40,z0,tPen\WObj:=wPaper;
    MoveL Offs(pOrigin,48.67,93.14,0.00),v40,z0,tPen\WObj:=wPaper;
    MoveL Offs(pOrigin,57.05,101.52,0.00),v40,z0,tPen\WObj:=wPaper;
    MoveL Offs(pOrigin,57.55,101.88,0.00),v40,z0,tPen\WObj:=wPaper;
    MoveL Offs(pOrigin,40.68,118.75,0.00),v40,z0,tPen\WObj:=wPaper;
    MoveL Offs(pOrigin,41.37,118.69,0.00),v40,z0,tPen\WObj:=wPaper;
    MoveL Offs(pOrigin,55.90,133.22,0.00),v40,z0,tPen\WObj:=wPaper;
    MoveL Offs(pOrigin,55.30,134.00,0.00),v40,z0,tPen\WObj:=wPaper;
    MoveL Offs(pOrigin,79.90,109.39,0.00),v40,z0,tPen\WObj:=wPaper;
    MoveL Offs(pOrigin,79.26,108.79,0.00),v40,z0,tPen\WObj:=wPaper;
    MoveL Offs(pOrigin,63.57,93.10,0.00),v40,z0,tPen\WObj:=wPaper;
    MoveL Offs(pOrigin,64.11,92.33,0.00),v40,z0,tPen\WObj:=wPaper;
    MoveL Offs(pOrigin,58.81,97.63,0.00),v40,z0,tPen\WObj:=wPaper;
    MoveL Offs(pOrigin,57.85,97.10,0.00),v40,z0,tPen\WObj:=wPaper;
    MoveL Offs(pOrigin,39.61,115.34,0.00),v40,fine,tPen\WObj:=wPaper;
    MoveL Offs(pOrigin,39.61,115.34,6.00),v60,z5,tPen\WObj:=wPaper;
    MoveL Offs(pOrigin,41.15,114.97,6.00),vTravel,z5,tPen\WObj:=wPaper;
    MoveL Offs(pOrigin,41.15,114.97,0.00),v60,z0,tPen\WObj:=wPaper;
    MoveL Offs(pOrigin,56.15,114.97,0.00),v40,z0,tPen\WObj:=wPaper;
    MoveL Offs(pOrigin,57.02,114.92,0.00),v40,z0,tPen\WObj:=wPaper;
    MoveL Offs(pOrigin,35.06,92.97,0.00),v40,z0,tPen\WObj:=wPaper;
    MoveL Offs(pOrigin,34.33,92.24,0.00),v40,z0,tPen\WObj:=wPaper;
    MoveL Offs(pOrigin,32.32,94.26,0.00),v40,z0,tPen\WObj:=wPaper;
    MoveL Offs(pOrigin,33.04,93.93,0.00),v40,z0,tPen\WObj:=wPaper;
    MoveL Offs(pOrigin,57.22,118.11,0.00),v40,z0,tPen\WObj:=wPaper;
    MoveL Offs(pOrigin,56.30,118.14,0.00),v40,z0,tPen\WObj:=wPaper;
    MoveL Offs(pOrigin,42.20,118.14,0.00),v40,z0,tPen\WObj:=wPaper;
    MoveL Offs(pOrigin,42.50,119.19,0.00),v40,z0,tPen\WObj:=wPaper;
    MoveL Offs(pOrigin,56.30,119.19,0.00),v40,z0,tPen\WObj:=wPaper;
    MoveL Offs(pOrigin,57.22,119.60,0.00),v40,z0,tPen\WObj:=wPaper;
    MoveL Offs(pOrigin,33.46,95.84,0.00),v40,z0,tPen\WObj:=wPaper;
    MoveL Offs(pOrigin,32.96,96.60,0.00),v40,z0,tPen\WObj:=wPaper;
    MoveL Offs(pOrigin,37.52,92.04,0.00),v40,z0,tPen\WObj:=wPaper;
    MoveL Offs(pOrigin,36.99,91.08,0.00),v40,z0,tPen\WObj:=wPaper;
    MoveL Offs(pOrigin,60.75,67.32,0.00),v40,z0,tPen\WObj:=wPaper;
    MoveL Offs(pOrigin,61.08,68.21,0.00),v40,z0,tPen\WObj:=wPaper;
    MoveL Offs(pOrigin,83.46,90.59,0.00),v40,fine,tPen\WObj:=wPaper;
    MoveL Offs(pOrigin,83.46,90.59,6.00),v60,z5,tPen\WObj:=wPaper;
    MoveL Offs(pOrigin,83.79,92.07,6.00),vTravel,z5,tPen\WObj:=wPaper;
    MoveL Offs(pOrigin,83.79,92.07,0.00),v60,z0,tPen\WObj:=wPaper;
    MoveL Offs(pOrigin,44.65,131.20,0.00),v40,fine,tPen\WObj:=wPaper;
    MoveL Offs(pOrigin,44.65,131.20,6.00),v60,z5,tPen\WObj:=wPaper;
    MoveL Offs(pOrigin,44.44,129.93,6.00),vTravel,z5,tPen\WObj:=wPaper;
    MoveL Offs(pOrigin,44.44,129.93,0.00),v60,z0,tPen\WObj:=wPaper;
    MoveL Offs(pOrigin,57.91,116.46,0.00),v40,z0,tPen\WObj:=wPaper;
    MoveL Offs(pOrigin,57.12,116.52,0.00),v40,z0,tPen\WObj:=wPaper;
    MoveL Offs(pOrigin,33.68,93.08,0.00),v40,z0,tPen\WObj:=wPaper;
    MoveL Offs(pOrigin,33.95,93.85,0.00),v40,z0,tPen\WObj:=wPaper;
    MoveL Offs(pOrigin,56.00,93.85,0.00),v40,z0,tPen\WObj:=wPaper;
    MoveL Offs(pOrigin,56.30,94.90,0.00),v40,z0,tPen\WObj:=wPaper;
    MoveL Offs(pOrigin,34.10,94.90,0.00),v40,z0,tPen\WObj:=wPaper;
    MoveL Offs(pOrigin,34.40,95.96,0.00),v40,z0,tPen\WObj:=wPaper;
    MoveL Offs(pOrigin,56.30,95.96,0.00),v40,z0,tPen\WObj:=wPaper;
    MoveL Offs(pOrigin,56.30,97.02,0.00),v40,z0,tPen\WObj:=wPaper;
    MoveL Offs(pOrigin,34.70,97.02,0.00),v40,z0,tPen\WObj:=wPaper;
    MoveL Offs(pOrigin,35.15,98.07,0.00),v40,z0,tPen\WObj:=wPaper;
    MoveL Offs(pOrigin,56.30,98.07,0.00),v40,z0,tPen\WObj:=wPaper;
    MoveL Offs(pOrigin,56.30,99.13,0.00),v40,z0,tPen\WObj:=wPaper;
    MoveL Offs(pOrigin,35.45,99.13,0.00),v40,fine,tPen\WObj:=wPaper;
    MoveL Offs(pOrigin,35.45,99.13,6.00),v60,z5,tPen\WObj:=wPaper;
    MoveL Offs(pOrigin,34.03,100.01,6.00),vTravel,z5,tPen\WObj:=wPaper;
    MoveL Offs(pOrigin,34.03,100.01,0.00),v60,z0,tPen\WObj:=wPaper;
    MoveL Offs(pOrigin,41.67,92.37,0.00),v40,z0,tPen\WObj:=wPaper;
    MoveL Offs(pOrigin,41.23,93.16,0.00),v40,z0,tPen\WObj:=wPaper;
    MoveL Offs(pOrigin,57.03,108.96,0.00),v40,z0,tPen\WObj:=wPaper;
    MoveL Offs(pOrigin,57.78,109.12,0.00),v40,z0,tPen\WObj:=wPaper;
    MoveL Offs(pOrigin,42.51,124.39,0.00),v40,z0,tPen\WObj:=wPaper;
    MoveL Offs(pOrigin,43.04,125.35,0.00),v40,z0,tPen\WObj:=wPaper;
    MoveL Offs(pOrigin,57.89,110.50,0.00),v40,fine,tPen\WObj:=wPaper;
    MoveL Offs(pOrigin,57.89,110.50,6.00),v60,z5,tPen\WObj:=wPaper;
    MoveL Offs(pOrigin,57.02,111.94,6.00),vTravel,z5,tPen\WObj:=wPaper;
    MoveL Offs(pOrigin,57.02,111.94,0.00),v60,z0,tPen\WObj:=wPaper;
    MoveL Offs(pOrigin,38.25,93.17,0.00),v40,z0,tPen\WObj:=wPaper;
    MoveL Offs(pOrigin,38.80,92.26,0.00),v40,z0,tPen\WObj:=wPaper;
    MoveL Offs(pOrigin,33.39,97.67,0.00),v40,fine,tPen\WObj:=wPaper;
    MoveL Offs(pOrigin,33.39,97.67,6.00),v60,z5,tPen\WObj:=wPaper;
    MoveL Offs(pOrigin,32.64,95.43,6.00),vTravel,z5,tPen\WObj:=wPaper;
    MoveL Offs(pOrigin,32.64,95.43,0.00),v60,z0,tPen\WObj:=wPaper;
    MoveL Offs(pOrigin,35.82,92.25,0.00),v40,fine,tPen\WObj:=wPaper;
    MoveL Offs(pOrigin,35.82,92.25,6.00),v60,z5,tPen\WObj:=wPaper;
    MoveL Offs(pOrigin,36.76,93.17,6.00),vTravel,z5,tPen\WObj:=wPaper;
    MoveL Offs(pOrigin,36.76,93.17,0.00),v60,z0,tPen\WObj:=wPaper;
    MoveL Offs(pOrigin,57.02,113.43,0.00),v40,z0,tPen\WObj:=wPaper;
    MoveL Offs(pOrigin,56.30,113.91,0.00),v40,z0,tPen\WObj:=wPaper;
    MoveL Offs(pOrigin,40.70,113.91,0.00),v40,z0,tPen\WObj:=wPaper;
    MoveL Offs(pOrigin,40.40,112.86,0.00),v40,z0,tPen\WObj:=wPaper;
    MoveL Offs(pOrigin,56.30,112.86,0.00),v40,z0,tPen\WObj:=wPaper;
    MoveL Offs(pOrigin,56.30,111.80,0.00),v40,z0,tPen\WObj:=wPaper;
    MoveL Offs(pOrigin,39.95,111.80,0.00),v40,fine,tPen\WObj:=wPaper;
    MoveL Offs(pOrigin,39.95,111.80,6.00),v60,z5,tPen\WObj:=wPaper;
  ENDPROC

  PROC DrawPart9()
    MoveL Offs(pOrigin,38.75,113.21,6.00),vTravel,z5,tPen\WObj:=wPaper;
    MoveL Offs(pOrigin,38.75,113.21,0.00),v60,z0,tPen\WObj:=wPaper;
    MoveL Offs(pOrigin,57.53,94.44,0.00),v40,fine,tPen\WObj:=wPaper;
    MoveL Offs(pOrigin,57.53,94.44,6.00),v60,z5,tPen\WObj:=wPaper;
    MoveL Offs(pOrigin,59.12,94.34,6.00),vTravel,z5,tPen\WObj:=wPaper;
    MoveL Offs(pOrigin,59.12,94.34,0.00),v60,z0,tPen\WObj:=wPaper;
    MoveL Offs(pOrigin,61.14,92.32,0.00),v40,fine,tPen\WObj:=wPaper;
    MoveL Offs(pOrigin,61.14,92.32,6.00),v60,z5,tPen\WObj:=wPaper;
    MoveL Offs(pOrigin,61.78,94.87,6.00),vTravel,z5,tPen\WObj:=wPaper;
    MoveL Offs(pOrigin,61.78,94.87,0.00),v60,z0,tPen\WObj:=wPaper;
    MoveL Offs(pOrigin,61.78,106.28,0.00),v40,fine,tPen\WObj:=wPaper;
    MoveL Offs(pOrigin,61.78,106.28,6.00),v60,z5,tPen\WObj:=wPaper;
    MoveL Offs(pOrigin,60.35,106.52,6.00),vTravel,z5,tPen\WObj:=wPaper;
    MoveL Offs(pOrigin,60.35,106.52,0.00),v60,z0,tPen\WObj:=wPaper;
    MoveL Offs(pOrigin,79.10,106.52,0.00),v40,z0,tPen\WObj:=wPaper;
    MoveL Offs(pOrigin,78.80,107.58,0.00),v40,z0,tPen\WObj:=wPaper;
    MoveL Offs(pOrigin,60.50,107.58,0.00),v40,z0,tPen\WObj:=wPaper;
    MoveL Offs(pOrigin,60.50,108.63,0.00),v40,z0,tPen\WObj:=wPaper;
    MoveL Offs(pOrigin,78.35,108.63,0.00),v40,fine,tPen\WObj:=wPaper;
    MoveL Offs(pOrigin,78.35,108.63,6.00),v60,z5,tPen\WObj:=wPaper;
    MoveL Offs(pOrigin,79.59,107.62,6.00),vTravel,z5,tPen\WObj:=wPaper;
    MoveL Offs(pOrigin,79.59,107.62,0.00),v60,z0,tPen\WObj:=wPaper;
    MoveL Offs(pOrigin,65.06,93.09,0.00),v40,fine,tPen\WObj:=wPaper;
    MoveL Offs(pOrigin,65.06,93.09,6.00),v60,z5,tPen\WObj:=wPaper;
    MoveL Offs(pOrigin,63.90,95.02,6.00),vTravel,z5,tPen\WObj:=wPaper;
    MoveL Offs(pOrigin,63.90,95.02,0.00),v60,z0,tPen\WObj:=wPaper;
    MoveL Offs(pOrigin,63.90,108.08,0.00),v40,z0,tPen\WObj:=wPaper;
    MoveL Offs(pOrigin,64.95,108.38,0.00),v40,z0,tPen\WObj:=wPaper;
    MoveL Offs(pOrigin,64.95,95.62,0.00),v40,fine,tPen\WObj:=wPaper;
    MoveL Offs(pOrigin,64.95,95.62,6.00),v60,z5,tPen\WObj:=wPaper;
    MoveL Offs(pOrigin,66.01,96.52,6.00),vTravel,z5,tPen\WObj:=wPaper;
    MoveL Offs(pOrigin,66.01,96.52,0.00),v60,z0,tPen\WObj:=wPaper;
    MoveL Offs(pOrigin,66.01,108.98,0.00),v40,fine,tPen\WObj:=wPaper;
    MoveL Offs(pOrigin,66.01,108.98,6.00),v60,z5,tPen\WObj:=wPaper;
    MoveL Offs(pOrigin,67.06,111.08,6.00),vTravel,z5,tPen\WObj:=wPaper;
    MoveL Offs(pOrigin,67.06,111.08,0.00),v60,z0,tPen\WObj:=wPaper;
    MoveL Offs(pOrigin,67.06,97.42,0.00),v40,fine,tPen\WObj:=wPaper;
    MoveL Offs(pOrigin,67.06,97.42,6.00),v60,z5,tPen\WObj:=wPaper;
    MoveL Offs(pOrigin,68.12,98.17,6.00),vTravel,z5,tPen\WObj:=wPaper;
    MoveL Offs(pOrigin,68.12,98.17,0.00),v60,z0,tPen\WObj:=wPaper;
    MoveL Offs(pOrigin,68.12,102.52,0.00),v40,z0,tPen\WObj:=wPaper;
    MoveL Offs(pOrigin,69.18,102.22,0.00),v40,z0,tPen\WObj:=wPaper;
    MoveL Offs(pOrigin,69.18,97.87,0.00),v40,fine,tPen\WObj:=wPaper;
    MoveL Offs(pOrigin,69.18,97.87,6.00),v60,z5,tPen\WObj:=wPaper;
    MoveL Offs(pOrigin,70.23,94.87,6.00),vTravel,z5,tPen\WObj:=wPaper;
    MoveL Offs(pOrigin,70.23,94.87,0.00),v60,z0,tPen\WObj:=wPaper;
    MoveL Offs(pOrigin,70.23,102.08,0.00),v40,fine,tPen\WObj:=wPaper;
    MoveL Offs(pOrigin,70.23,102.08,6.00),v60,z5,tPen\WObj:=wPaper;
    MoveL Offs(pOrigin,71.29,102.82,6.00),vTravel,z5,tPen\WObj:=wPaper;
    MoveL Offs(pOrigin,71.29,102.82,0.00),v60,z0,tPen\WObj:=wPaper;
    MoveL Offs(pOrigin,71.29,94.87,0.00),v40,z0,tPen\WObj:=wPaper;
    MoveL Offs(pOrigin,72.34,94.87,0.00),v40,z0,tPen\WObj:=wPaper;
    MoveL Offs(pOrigin,72.34,104.02,0.00),v40,fine,tPen\WObj:=wPaper;
    MoveL Offs(pOrigin,72.34,104.02,6.00),v60,z5,tPen\WObj:=wPaper;
    MoveL Offs(pOrigin,73.40,104.92,6.00),vTravel,z5,tPen\WObj:=wPaper;
    MoveL Offs(pOrigin,73.40,104.92,0.00),v60,z0,tPen\WObj:=wPaper;
    MoveL Offs(pOrigin,73.40,94.87,0.00),v40,z0,tPen\WObj:=wPaper;
    MoveL Offs(pOrigin,74.46,94.87,0.00),v40,z0,tPen\WObj:=wPaper;
    MoveL Offs(pOrigin,74.46,105.52,0.00),v40,fine,tPen\WObj:=wPaper;
    MoveL Offs(pOrigin,74.46,105.52,6.00),v60,z5,tPen\WObj:=wPaper;
    MoveL Offs(pOrigin,75.51,106.42,6.00),vTravel,z5,tPen\WObj:=wPaper;
    MoveL Offs(pOrigin,75.51,106.42,0.00),v60,z0,tPen\WObj:=wPaper;
    MoveL Offs(pOrigin,75.51,94.87,0.00),v40,z0,tPen\WObj:=wPaper;
    MoveL Offs(pOrigin,76.57,94.87,0.00),v40,z0,tPen\WObj:=wPaper;
    MoveL Offs(pOrigin,76.57,107.78,0.00),v40,fine,tPen\WObj:=wPaper;
    MoveL Offs(pOrigin,76.57,107.78,6.00),v60,z5,tPen\WObj:=wPaper;
    MoveL Offs(pOrigin,77.62,106.28,6.00),vTravel,z5,tPen\WObj:=wPaper;
    MoveL Offs(pOrigin,77.62,106.28,0.00),v60,z0,tPen\WObj:=wPaper;
    MoveL Offs(pOrigin,77.62,95.48,0.00),v40,fine,tPen\WObj:=wPaper;
    MoveL Offs(pOrigin,77.62,95.48,6.00),v60,z5,tPen\WObj:=wPaper;
    MoveL Offs(pOrigin,78.68,96.37,6.00),vTravel,z5,tPen\WObj:=wPaper;
    MoveL Offs(pOrigin,78.68,96.37,0.00),v60,z0,tPen\WObj:=wPaper;
    MoveL Offs(pOrigin,78.68,103.72,0.00),v40,fine,tPen\WObj:=wPaper;
    MoveL Offs(pOrigin,78.68,103.72,6.00),v60,z5,tPen\WObj:=wPaper;
    MoveL Offs(pOrigin,79.55,105.46,6.00),vTravel,z5,tPen\WObj:=wPaper;
    MoveL Offs(pOrigin,79.55,105.46,0.00),v60,z0,tPen\WObj:=wPaper;
    MoveL Offs(pOrigin,60.35,105.46,0.00),v40,fine,tPen\WObj:=wPaper;
    MoveL Offs(pOrigin,60.35,105.46,6.00),v60,z5,tPen\WObj:=wPaper;
    MoveL Offs(pOrigin,58.95,107.95,6.00),vTravel,z5,tPen\WObj:=wPaper;
    MoveL Offs(pOrigin,58.95,107.95,0.00),v60,z0,tPen\WObj:=wPaper;
    MoveL Offs(pOrigin,74.96,91.93,0.00),v40,z0,tPen\WObj:=wPaper;
    MoveL Offs(pOrigin,75.37,92.96,0.00),v40,z0,tPen\WObj:=wPaper;
    MoveL Offs(pOrigin,82.37,99.96,0.00),v40,z0,tPen\WObj:=wPaper;
    MoveL Offs(pOrigin,83.39,99.94,0.00),v40,z0,tPen\WObj:=wPaper;
    MoveL Offs(pOrigin,49.34,133.98,0.00),v40,z0,tPen\WObj:=wPaper;
    MoveL Offs(pOrigin,50.05,133.34,0.00),v40,z0,tPen\WObj:=wPaper;
    MoveL Offs(pOrigin,44.32,127.62,0.00),v40,z0,tPen\WObj:=wPaper;
    MoveL Offs(pOrigin,45.35,127.64,0.00),v40,z0,tPen\WObj:=wPaper;
    MoveL Offs(pOrigin,56.45,127.64,0.00),v40,z0,tPen\WObj:=wPaper;
    MoveL Offs(pOrigin,57.19,127.05,0.00),v40,z0,tPen\WObj:=wPaper;
    MoveL Offs(pOrigin,37.47,107.32,0.00),v40,z0,tPen\WObj:=wPaper;
    MoveL Offs(pOrigin,38.00,106.52,0.00),v40,z0,tPen\WObj:=wPaper;
    MoveL Offs(pOrigin,56.30,106.52,0.00),v40,z0,tPen\WObj:=wPaper;
    MoveL Offs(pOrigin,56.30,105.46,0.00),v40,z0,tPen\WObj:=wPaper;
    MoveL Offs(pOrigin,37.70,105.46,0.00),v40,z0,tPen\WObj:=wPaper;
    MoveL Offs(pOrigin,37.40,104.41,0.00),v40,z0,tPen\WObj:=wPaper;
    MoveL Offs(pOrigin,56.30,104.41,0.00),v40,z0,tPen\WObj:=wPaper;
    MoveL Offs(pOrigin,56.30,103.35,0.00),v40,z0,tPen\WObj:=wPaper;
    MoveL Offs(pOrigin,36.95,103.35,0.00),v40,z0,tPen\WObj:=wPaper;
    MoveL Offs(pOrigin,36.50,102.30,0.00),v40,z0,tPen\WObj:=wPaper;
    MoveL Offs(pOrigin,56.30,102.30,0.00),v40,z0,tPen\WObj:=wPaper;
    MoveL Offs(pOrigin,57.05,103.01,0.00),v40,z0,tPen\WObj:=wPaper;
    MoveL Offs(pOrigin,47.19,93.14,0.00),v40,z0,tPen\WObj:=wPaper;
    MoveL Offs(pOrigin,47.63,92.39,0.00),v40,z0,tPen\WObj:=wPaper;
    MoveL Offs(pOrigin,35.85,104.16,0.00),v40,fine,tPen\WObj:=wPaper;
    MoveL Offs(pOrigin,35.85,104.16,6.00),v60,z5,tPen\WObj:=wPaper;
    MoveL Offs(pOrigin,36.20,101.24,6.00),vTravel,z5,tPen\WObj:=wPaper;
    MoveL Offs(pOrigin,36.20,101.24,0.00),v60,z0,tPen\WObj:=wPaper;
    MoveL Offs(pOrigin,56.30,101.24,0.00),v40,fine,tPen\WObj:=wPaper;
    MoveL Offs(pOrigin,56.30,101.24,6.00),v60,z5,tPen\WObj:=wPaper;
    MoveL Offs(pOrigin,57.65,100.29,6.00),vTravel,z5,tPen\WObj:=wPaper;
    MoveL Offs(pOrigin,57.65,100.29,0.00),v60,z0,tPen\WObj:=wPaper;
    MoveL Offs(pOrigin,40.25,117.68,0.00),v40,fine,tPen\WObj:=wPaper;
    MoveL Offs(pOrigin,40.25,117.68,6.00),v60,z5,tPen\WObj:=wPaper;
    MoveL Offs(pOrigin,41.75,117.08,6.00),vTravel,z5,tPen\WObj:=wPaper;
    MoveL Offs(pOrigin,41.75,117.08,0.00),v60,z0,tPen\WObj:=wPaper;
    MoveL Offs(pOrigin,56.30,117.08,0.00),v40,z0,tPen\WObj:=wPaper;
    MoveL Offs(pOrigin,56.30,116.02,0.00),v40,z0,tPen\WObj:=wPaper;
    MoveL Offs(pOrigin,41.45,116.02,0.00),v40,fine,tPen\WObj:=wPaper;
    MoveL Offs(pOrigin,41.45,116.02,6.00),v60,z5,tPen\WObj:=wPaper;
  ENDPROC

  PROC DrawPart10()
    MoveL Offs(pOrigin,44.89,116.48,6.00),vTravel,z5,tPen\WObj:=wPaper;
    MoveL Offs(pOrigin,44.89,116.48,0.00),v60,z0,tPen\WObj:=wPaper;
    MoveL Offs(pOrigin,44.89,120.37,0.00),v40,fine,tPen\WObj:=wPaper;
    MoveL Offs(pOrigin,44.89,120.37,6.00),v60,z5,tPen\WObj:=wPaper;
    MoveL Offs(pOrigin,42.80,120.25,6.00),vTravel,z5,tPen\WObj:=wPaper;
    MoveL Offs(pOrigin,42.80,120.25,0.00),v60,z0,tPen\WObj:=wPaper;
    MoveL Offs(pOrigin,56.30,120.25,0.00),v40,fine,tPen\WObj:=wPaper;
    MoveL Offs(pOrigin,56.30,120.25,6.00),v60,z5,tPen\WObj:=wPaper;
    MoveL Offs(pOrigin,56.30,123.42,6.00),vTravel,z5,tPen\WObj:=wPaper;
    MoveL Offs(pOrigin,56.30,123.42,0.00),v60,z0,tPen\WObj:=wPaper;
    MoveL Offs(pOrigin,44.00,123.42,0.00),v40,fine,tPen\WObj:=wPaper;
    MoveL Offs(pOrigin,44.00,123.42,6.00),v60,z5,tPen\WObj:=wPaper;
    MoveL Offs(pOrigin,43.58,125.38,6.00),vTravel,z5,tPen\WObj:=wPaper;
    MoveL Offs(pOrigin,43.58,125.38,0.00),v60,z0,tPen\WObj:=wPaper;
    MoveL Offs(pOrigin,51.54,133.34,0.00),v40,z0,tPen\WObj:=wPaper;
    MoveL Offs(pOrigin,50.83,133.99,0.00),v40,z0,tPen\WObj:=wPaper;
    MoveL Offs(pOrigin,82.44,102.38,0.00),v40,fine,tPen\WObj:=wPaper;
    MoveL Offs(pOrigin,82.44,102.38,6.00),v60,z5,tPen\WObj:=wPaper;
    MoveL Offs(pOrigin,80.75,102.30,6.00),vTravel,z5,tPen\WObj:=wPaper;
    MoveL Offs(pOrigin,80.75,102.30,0.00),v60,z0,tPen\WObj:=wPaper;
    MoveL Offs(pOrigin,60.35,102.30,0.00),v40,fine,tPen\WObj:=wPaper;
    MoveL Offs(pOrigin,60.35,102.30,6.00),v60,z5,tPen\WObj:=wPaper;
    MoveL Offs(pOrigin,59.03,100.40,6.00),vTravel,z5,tPen\WObj:=wPaper;
    MoveL Offs(pOrigin,59.03,100.40,0.00),v60,z0,tPen\WObj:=wPaper;
    MoveL Offs(pOrigin,67.41,92.02,0.00),v40,z0,tPen\WObj:=wPaper;
    MoveL Offs(pOrigin,67.82,92.87,0.00),v40,z0,tPen\WObj:=wPaper;
    MoveL Offs(pOrigin,80.44,105.49,0.00),v40,fine,tPen\WObj:=wPaper;
    MoveL Offs(pOrigin,80.44,105.49,6.00),v60,z5,tPen\WObj:=wPaper;
    MoveL Offs(pOrigin,81.81,104.51,6.00),vTravel,z5,tPen\WObj:=wPaper;
    MoveL Offs(pOrigin,81.81,104.51,0.00),v60,z0,tPen\WObj:=wPaper;
    MoveL Offs(pOrigin,52.11,134.20,0.00),v40,fine,tPen\WObj:=wPaper;
    MoveL Offs(pOrigin,52.11,134.20,6.00),v60,z5,tPen\WObj:=wPaper;
    MoveL Offs(pOrigin,54.52,133.33,6.00),vTravel,z5,tPen\WObj:=wPaper;
    MoveL Offs(pOrigin,54.52,133.33,0.00),v60,z0,tPen\WObj:=wPaper;
    MoveL Offs(pOrigin,42.11,120.92,0.00),v40,fine,tPen\WObj:=wPaper;
    MoveL Offs(pOrigin,42.11,120.92,6.00),v60,z5,tPen\WObj:=wPaper;
    MoveL Offs(pOrigin,41.00,119.92,6.00),vTravel,z5,tPen\WObj:=wPaper;
    MoveL Offs(pOrigin,41.00,119.92,0.00),v60,z0,tPen\WObj:=wPaper;
    MoveL Offs(pOrigin,57.76,103.16,0.00),v40,fine,tPen\WObj:=wPaper;
    MoveL Offs(pOrigin,57.76,103.16,6.00),v60,z5,tPen\WObj:=wPaper;
    MoveL Offs(pOrigin,56.30,107.58,6.00),vTravel,z5,tPen\WObj:=wPaper;
    MoveL Offs(pOrigin,56.30,107.58,0.00),v60,z0,tPen\WObj:=wPaper;
    MoveL Offs(pOrigin,38.45,107.58,0.00),v40,z0,tPen\WObj:=wPaper;
    MoveL Offs(pOrigin,38.75,108.63,0.00),v40,z0,tPen\WObj:=wPaper;
    MoveL Offs(pOrigin,56.30,108.63,0.00),v40,z0,tPen\WObj:=wPaper;
    MoveL Offs(pOrigin,56.30,109.69,0.00),v40,z0,tPen\WObj:=wPaper;
    MoveL Offs(pOrigin,39.20,109.69,0.00),v40,fine,tPen\WObj:=wPaper;
    MoveL Offs(pOrigin,39.20,109.69,6.00),v60,z5,tPen\WObj:=wPaper;
    MoveL Offs(pOrigin,37.36,108.63,6.00),vTravel,z5,tPen\WObj:=wPaper;
    MoveL Offs(pOrigin,37.36,108.63,0.00),v60,z0,tPen\WObj:=wPaper;
    MoveL Offs(pOrigin,53.58,92.41,0.00),v40,z0,tPen\WObj:=wPaper;
    MoveL Offs(pOrigin,53.14,93.13,0.00),v40,z0,tPen\WObj:=wPaper;
    MoveL Offs(pOrigin,57.07,97.05,0.00),v40,fine,tPen\WObj:=wPaper;
    MoveL Offs(pOrigin,57.07,97.05,6.00),v60,z5,tPen\WObj:=wPaper;
    MoveL Offs(pOrigin,54.39,97.57,6.00),vTravel,z5,tPen\WObj:=wPaper;
    MoveL Offs(pOrigin,54.39,97.57,0.00),v60,z0,tPen\WObj:=wPaper;
    MoveL Offs(pOrigin,54.39,112.42,0.00),v40,fine,tPen\WObj:=wPaper;
    MoveL Offs(pOrigin,54.39,112.42,6.00),v60,z5,tPen\WObj:=wPaper;
    MoveL Offs(pOrigin,53.34,110.62,6.00),vTravel,z5,tPen\WObj:=wPaper;
    MoveL Offs(pOrigin,53.34,110.62,0.00),v60,z0,tPen\WObj:=wPaper;
    MoveL Offs(pOrigin,53.34,96.67,0.00),v40,fine,tPen\WObj:=wPaper;
    MoveL Offs(pOrigin,53.34,96.67,6.00),v60,z5,tPen\WObj:=wPaper;
    MoveL Offs(pOrigin,52.28,95.62,6.00),vTravel,z5,tPen\WObj:=wPaper;
    MoveL Offs(pOrigin,52.28,95.62,0.00),v60,z0,tPen\WObj:=wPaper;
    MoveL Offs(pOrigin,52.28,109.42,0.00),v40,z0,tPen\WObj:=wPaper;
    MoveL Offs(pOrigin,51.22,109.12,0.00),v40,z0,tPen\WObj:=wPaper;
    MoveL Offs(pOrigin,51.22,95.02,0.00),v40,z0,tPen\WObj:=wPaper;
    MoveL Offs(pOrigin,50.17,94.87,0.00),v40,z0,tPen\WObj:=wPaper;
    MoveL Offs(pOrigin,50.17,109.28,0.00),v40,fine,tPen\WObj:=wPaper;
    MoveL Offs(pOrigin,50.17,109.28,6.00),v60,z5,tPen\WObj:=wPaper;
    MoveL Offs(pOrigin,49.11,107.32,6.00),vTravel,z5,tPen\WObj:=wPaper;
    MoveL Offs(pOrigin,49.11,107.32,0.00),v60,z0,tPen\WObj:=wPaper;
    MoveL Offs(pOrigin,49.11,94.87,0.00),v40,z0,tPen\WObj:=wPaper;
    MoveL Offs(pOrigin,48.06,94.72,0.00),v40,z0,tPen\WObj:=wPaper;
    MoveL Offs(pOrigin,48.06,105.98,0.00),v40,fine,tPen\WObj:=wPaper;
    MoveL Offs(pOrigin,48.06,105.98,6.00),v60,z5,tPen\WObj:=wPaper;
    MoveL Offs(pOrigin,47.00,104.62,6.00),vTravel,z5,tPen\WObj:=wPaper;
    MoveL Offs(pOrigin,47.00,104.62,0.00),v60,z0,tPen\WObj:=wPaper;
    MoveL Offs(pOrigin,47.00,94.87,0.00),v40,z0,tPen\WObj:=wPaper;
    MoveL Offs(pOrigin,45.94,94.87,0.00),v40,z0,tPen\WObj:=wPaper;
    MoveL Offs(pOrigin,45.94,103.72,0.00),v40,fine,tPen\WObj:=wPaper;
    MoveL Offs(pOrigin,45.94,103.72,6.00),v60,z5,tPen\WObj:=wPaper;
    MoveL Offs(pOrigin,44.89,102.38,6.00),vTravel,z5,tPen\WObj:=wPaper;
    MoveL Offs(pOrigin,44.89,102.38,0.00),v60,z0,tPen\WObj:=wPaper;
    MoveL Offs(pOrigin,44.89,95.02,0.00),v40,fine,tPen\WObj:=wPaper;
    MoveL Offs(pOrigin,44.89,95.02,6.00),v60,z5,tPen\WObj:=wPaper;
    MoveL Offs(pOrigin,43.83,97.57,6.00),vTravel,z5,tPen\WObj:=wPaper;
    MoveL Offs(pOrigin,43.83,97.57,0.00),v60,z0,tPen\WObj:=wPaper;
    MoveL Offs(pOrigin,43.83,101.78,0.00),v40,z0,tPen\WObj:=wPaper;
    MoveL Offs(pOrigin,42.78,102.08,0.00),v40,z0,tPen\WObj:=wPaper;
    MoveL Offs(pOrigin,42.78,98.62,0.00),v40,z0,tPen\WObj:=wPaper;
    MoveL Offs(pOrigin,41.72,98.48,0.00),v40,z0,tPen\WObj:=wPaper;
    MoveL Offs(pOrigin,41.72,102.22,0.00),v40,fine,tPen\WObj:=wPaper;
    MoveL Offs(pOrigin,41.72,102.22,6.00),v60,z5,tPen\WObj:=wPaper;
    MoveL Offs(pOrigin,41.72,105.08,6.00),vTravel,z5,tPen\WObj:=wPaper;
    MoveL Offs(pOrigin,41.72,105.08,0.00),v60,z0,tPen\WObj:=wPaper;
    MoveL Offs(pOrigin,41.72,108.52,0.00),v40,fine,tPen\WObj:=wPaper;
    MoveL Offs(pOrigin,41.72,108.52,6.00),v60,z5,tPen\WObj:=wPaper;
    MoveL Offs(pOrigin,42.78,107.32,6.00),vTravel,z5,tPen\WObj:=wPaper;
    MoveL Offs(pOrigin,42.78,107.32,0.00),v60,z0,tPen\WObj:=wPaper;
    MoveL Offs(pOrigin,42.78,110.62,0.00),v40,fine,tPen\WObj:=wPaper;
    MoveL Offs(pOrigin,42.78,110.62,6.00),v60,z5,tPen\WObj:=wPaper;
    MoveL Offs(pOrigin,43.83,112.58,6.00),vTravel,z5,tPen\WObj:=wPaper;
    MoveL Offs(pOrigin,43.83,112.58,0.00),v60,z0,tPen\WObj:=wPaper;
    MoveL Offs(pOrigin,43.83,107.62,0.00),v40,z0,tPen\WObj:=wPaper;
    MoveL Offs(pOrigin,44.89,107.62,0.00),v40,z0,tPen\WObj:=wPaper;
    MoveL Offs(pOrigin,44.89,113.18,0.00),v40,fine,tPen\WObj:=wPaper;
    MoveL Offs(pOrigin,44.89,113.18,6.00),v60,z5,tPen\WObj:=wPaper;
    MoveL Offs(pOrigin,48.06,110.92,6.00),vTravel,z5,tPen\WObj:=wPaper;
    MoveL Offs(pOrigin,48.06,110.92,0.00),v60,z0,tPen\WObj:=wPaper;
    MoveL Offs(pOrigin,48.06,124.72,0.00),v40,fine,tPen\WObj:=wPaper;
    MoveL Offs(pOrigin,48.06,124.72,6.00),v60,z5,tPen\WObj:=wPaper;
    MoveL Offs(pOrigin,49.11,126.07,6.00),vTravel,z5,tPen\WObj:=wPaper;
    MoveL Offs(pOrigin,49.11,126.07,0.00),v60,z0,tPen\WObj:=wPaper;
    MoveL Offs(pOrigin,49.11,111.82,0.00),v40,fine,tPen\WObj:=wPaper;
    MoveL Offs(pOrigin,49.11,111.82,6.00),v60,z5,tPen\WObj:=wPaper;
    MoveL Offs(pOrigin,50.17,113.02,6.00),vTravel,z5,tPen\WObj:=wPaper;
    MoveL Offs(pOrigin,50.17,113.02,0.00),v60,z0,tPen\WObj:=wPaper;
    MoveL Offs(pOrigin,50.17,127.87,0.00),v40,z0,tPen\WObj:=wPaper;
    MoveL Offs(pOrigin,51.22,128.32,0.00),v40,z0,tPen\WObj:=wPaper;
  ENDPROC

  PROC DrawPart11()
    MoveL Offs(pOrigin,51.22,114.08,0.00),v40,fine,tPen\WObj:=wPaper;
    MoveL Offs(pOrigin,51.22,114.08,6.00),v60,z5,tPen\WObj:=wPaper;
    MoveL Offs(pOrigin,52.28,115.12,6.00),vTravel,z5,tPen\WObj:=wPaper;
    MoveL Offs(pOrigin,52.28,115.12,0.00),v60,z0,tPen\WObj:=wPaper;
    MoveL Offs(pOrigin,52.28,128.77,0.00),v40,fine,tPen\WObj:=wPaper;
    MoveL Offs(pOrigin,52.28,128.77,6.00),v60,z5,tPen\WObj:=wPaper;
    MoveL Offs(pOrigin,53.34,130.57,6.00),vTravel,z5,tPen\WObj:=wPaper;
    MoveL Offs(pOrigin,53.34,130.57,0.00),v60,z0,tPen\WObj:=wPaper;
    MoveL Offs(pOrigin,53.34,116.02,0.00),v40,fine,tPen\WObj:=wPaper;
    MoveL Offs(pOrigin,53.34,116.02,6.00),v60,z5,tPen\WObj:=wPaper;
    MoveL Offs(pOrigin,54.39,117.22,6.00),vTravel,z5,tPen\WObj:=wPaper;
    MoveL Offs(pOrigin,54.39,117.22,0.00),v60,z0,tPen\WObj:=wPaper;
    MoveL Offs(pOrigin,54.39,130.88,0.00),v40,fine,tPen\WObj:=wPaper;
    MoveL Offs(pOrigin,54.39,130.88,6.00),v60,z5,tPen\WObj:=wPaper;
    MoveL Offs(pOrigin,56.45,130.81,6.00),vTravel,z5,tPen\WObj:=wPaper;
    MoveL Offs(pOrigin,56.45,130.81,0.00),v60,z0,tPen\WObj:=wPaper;
    MoveL Offs(pOrigin,46.40,130.81,0.00),v40,fine,tPen\WObj:=wPaper;
    MoveL Offs(pOrigin,46.40,130.81,6.00),v60,z5,tPen\WObj:=wPaper;
    MoveL Offs(pOrigin,45.27,130.06,6.00),vTravel,z5,tPen\WObj:=wPaper;
    MoveL Offs(pOrigin,45.27,130.06,0.00),v60,z0,tPen\WObj:=wPaper;
    MoveL Offs(pOrigin,48.56,133.35,0.00),v40,z0,tPen\WObj:=wPaper;
    MoveL Offs(pOrigin,47.85,133.98,0.00),v40,z0,tPen\WObj:=wPaper;
    MoveL Offs(pOrigin,83.60,98.23,0.00),v40,fine,tPen\WObj:=wPaper;
    MoveL Offs(pOrigin,83.60,98.23,6.00),v60,z5,tPen\WObj:=wPaper;
    MoveL Offs(pOrigin,82.55,97.02,6.00),vTravel,z5,tPen\WObj:=wPaper;
    MoveL Offs(pOrigin,82.55,97.02,0.00),v60,z0,tPen\WObj:=wPaper;
    MoveL Offs(pOrigin,60.35,97.02,0.00),v40,fine,tPen\WObj:=wPaper;
    MoveL Offs(pOrigin,60.35,97.02,6.00),v60,z5,tPen\WObj:=wPaper;
    MoveL Offs(pOrigin,62.84,94.87,6.00),vTravel,z5,tPen\WObj:=wPaper;
    MoveL Offs(pOrigin,62.84,94.87,0.00),v60,z0,tPen\WObj:=wPaper;
    MoveL Offs(pOrigin,62.84,107.78,0.00),v40,fine,tPen\WObj:=wPaper;
    MoveL Offs(pOrigin,62.84,107.78,6.00),v60,z5,tPen\WObj:=wPaper;
    MoveL Offs(pOrigin,59.69,108.64,6.00),vTravel,z5,tPen\WObj:=wPaper;
    MoveL Offs(pOrigin,59.69,108.64,0.00),v60,z0,tPen\WObj:=wPaper;
    MoveL Offs(pOrigin,74.22,123.17,0.00),v40,z0,tPen\WObj:=wPaper;
    MoveL Offs(pOrigin,75.26,123.00,0.00),v40,z0,tPen\WObj:=wPaper;
    MoveL Offs(pOrigin,64.13,134.13,0.00),v40,fine,tPen\WObj:=wPaper;
    MoveL Offs(pOrigin,64.13,134.13,6.00),v60,z5,tPen\WObj:=wPaper;
    MoveL Offs(pOrigin,63.35,133.20,6.00),vTravel,z5,tPen\WObj:=wPaper;
    MoveL Offs(pOrigin,63.35,133.20,0.00),v60,z0,tPen\WObj:=wPaper;
    MoveL Offs(pOrigin,59.53,129.38,0.00),v40,fine,tPen\WObj:=wPaper;
    MoveL Offs(pOrigin,59.53,129.38,6.00),v60,z5,tPen\WObj:=wPaper;
    MoveL Offs(pOrigin,59.42,130.76,6.00),vTravel,z5,tPen\WObj:=wPaper;
    MoveL Offs(pOrigin,59.42,130.76,0.00),v60,z0,tPen\WObj:=wPaper;
    MoveL Offs(pOrigin,61.96,133.31,0.00),v40,z0,tPen\WObj:=wPaper;
    MoveL Offs(pOrigin,62.85,133.92,0.00),v40,z0,tPen\WObj:=wPaper;
    MoveL Offs(pOrigin,76.00,120.76,0.00),v40,fine,tPen\WObj:=wPaper;
    MoveL Offs(pOrigin,76.00,120.76,6.00),v60,z5,tPen\WObj:=wPaper;
    MoveL Offs(pOrigin,70.70,130.81,6.00),vTravel,z5,tPen\WObj:=wPaper;
    MoveL Offs(pOrigin,70.70,130.81,0.00),v60,z0,tPen\WObj:=wPaper;
    MoveL Offs(pOrigin,60.35,130.81,0.00),v40,fine,tPen\WObj:=wPaper;
    MoveL Offs(pOrigin,60.35,130.81,6.00),v60,z5,tPen\WObj:=wPaper;
    MoveL Offs(pOrigin,63.90,126.97,6.00),vTravel,z5,tPen\WObj:=wPaper;
    MoveL Offs(pOrigin,63.90,126.97,0.00),v60,z0,tPen\WObj:=wPaper;
    MoveL Offs(pOrigin,63.90,122.77,0.00),v40,fine,tPen\WObj:=wPaper;
    MoveL Offs(pOrigin,63.90,122.77,6.00),v60,z5,tPen\WObj:=wPaper;
    MoveL Offs(pOrigin,61.78,123.97,6.00),vTravel,z5,tPen\WObj:=wPaper;
    MoveL Offs(pOrigin,61.78,123.97,0.00),v60,z0,tPen\WObj:=wPaper;
    MoveL Offs(pOrigin,61.78,112.58,0.00),v40,fine,tPen\WObj:=wPaper;
    MoveL Offs(pOrigin,61.78,112.58,6.00),v60,z5,tPen\WObj:=wPaper;
    MoveL Offs(pOrigin,57.80,115.07,6.00),vTravel,z5,tPen\WObj:=wPaper;
    MoveL Offs(pOrigin,57.80,115.07,0.00),v60,z0,tPen\WObj:=wPaper;
    MoveL Offs(pOrigin,44.11,128.76,0.00),v40,fine,tPen\WObj:=wPaper;
    MoveL Offs(pOrigin,44.11,128.76,6.00),v60,z5,tPen\WObj:=wPaper;
    MoveL Offs(pOrigin,45.05,126.58,6.00),vTravel,z5,tPen\WObj:=wPaper;
    MoveL Offs(pOrigin,45.05,126.58,0.00),v60,z0,tPen\WObj:=wPaper;
    MoveL Offs(pOrigin,56.30,126.58,0.00),v40,fine,tPen\WObj:=wPaper;
    MoveL Offs(pOrigin,56.30,126.58,6.00),v60,z5,tPen\WObj:=wPaper;
    MoveL Offs(pOrigin,62.84,125.17,6.00),vTravel,z5,tPen\WObj:=wPaper;
    MoveL Offs(pOrigin,62.84,125.17,0.00),v60,z0,tPen\WObj:=wPaper;
    MoveL Offs(pOrigin,62.84,117.97,0.00),v40,fine,tPen\WObj:=wPaper;
    MoveL Offs(pOrigin,62.84,117.97,6.00),v60,z5,tPen\WObj:=wPaper;
    MoveL Offs(pOrigin,68.12,111.22,6.00),vTravel,z5,tPen\WObj:=wPaper;
    MoveL Offs(pOrigin,68.12,111.22,0.00),v60,z0,tPen\WObj:=wPaper;
    MoveL Offs(pOrigin,68.12,104.92,0.00),v40,fine,tPen\WObj:=wPaper;
    MoveL Offs(pOrigin,68.12,104.92,6.00),v60,z5,tPen\WObj:=wPaper;
    MoveL Offs(pOrigin,69.18,107.48,6.00),vTravel,z5,tPen\WObj:=wPaper;
    MoveL Offs(pOrigin,69.18,107.48,0.00),v60,z0,tPen\WObj:=wPaper;
    MoveL Offs(pOrigin,69.18,110.78,0.00),v40,z0,tPen\WObj:=wPaper;
    MoveL Offs(pOrigin,70.23,110.32,0.00),v40,z0,tPen\WObj:=wPaper;
    MoveL Offs(pOrigin,70.23,108.08,0.00),v40,fine,tPen\WObj:=wPaper;
    MoveL Offs(pOrigin,70.23,108.08,6.00),v60,z5,tPen\WObj:=wPaper;
    MoveL Offs(pOrigin,71.29,108.82,6.00),vTravel,z5,tPen\WObj:=wPaper;
    MoveL Offs(pOrigin,71.29,108.82,0.00),v60,z0,tPen\WObj:=wPaper;
    MoveL Offs(pOrigin,71.29,110.02,0.00),v40,fine,tPen\WObj:=wPaper;
    MoveL Offs(pOrigin,71.29,110.02,6.00),v60,z5,tPen\WObj:=wPaper;
    MoveL Offs(pOrigin,79.74,101.17,6.00),vTravel,z5,tPen\WObj:=wPaper;
    MoveL Offs(pOrigin,79.74,101.17,0.00),v60,z0,tPen\WObj:=wPaper;
    MoveL Offs(pOrigin,79.74,97.28,0.00),v40,fine,tPen\WObj:=wPaper;
    MoveL Offs(pOrigin,79.74,97.28,6.00),v60,z5,tPen\WObj:=wPaper;
    MoveL Offs(pOrigin,85.18,93.67,6.00),vTravel,z5,tPen\WObj:=wPaper;
    MoveL Offs(pOrigin,85.18,93.67,0.00),v60,z0,tPen\WObj:=wPaper;
    MoveL Offs(pOrigin,45.40,133.44,0.00),v40,z0,tPen\WObj:=wPaper;
    MoveL Offs(pOrigin,44.87,132.48,0.00),v40,z0,tPen\WObj:=wPaper;
    MoveL Offs(pOrigin,84.75,92.60,0.00),v40,fine,tPen\WObj:=wPaper;
    MoveL Offs(pOrigin,84.75,92.60,6.00),v60,z5,tPen\WObj:=wPaper;
    MoveL Offs(pOrigin,85.40,88.57,6.00),vTravel,z5,tPen\WObj:=wPaper;
    MoveL Offs(pOrigin,85.40,88.57,0.00),v60,z0,tPen\WObj:=wPaper;
    MoveL Offs(pOrigin,60.65,88.57,0.00),v40,fine,tPen\WObj:=wPaper;
    MoveL Offs(pOrigin,60.65,88.57,6.00),v60,z5,tPen\WObj:=wPaper;
    MoveL Offs(pOrigin,64.00,90.95,6.00),vTravel,z5,tPen\WObj:=wPaper;
    MoveL Offs(pOrigin,64.00,90.95,0.00),v60,z0,tPen\WObj:=wPaper;
    MoveL Offs(pOrigin,98.58,56.37,0.00),v40,fine,tPen\WObj:=wPaper;
    MoveL Offs(pOrigin,98.58,56.37,6.00),v60,z5,tPen\WObj:=wPaper;
    MoveL Offs(pOrigin,98.25,54.60,6.00),vTravel,z5,tPen\WObj:=wPaper;
    MoveL Offs(pOrigin,98.25,54.60,0.00),v60,z0,tPen\WObj:=wPaper;
    MoveL Offs(pOrigin,94.32,50.67,0.00),v40,fine,tPen\WObj:=wPaper;
    MoveL Offs(pOrigin,94.32,50.67,6.00),v60,z5,tPen\WObj:=wPaper;
    MoveL Offs(pOrigin,97.40,54.78,6.00),vTravel,z5,tPen\WObj:=wPaper;
    MoveL Offs(pOrigin,97.40,54.78,0.00),v60,z0,tPen\WObj:=wPaper;
    MoveL Offs(pOrigin,78.50,54.78,0.00),v40,fine,tPen\WObj:=wPaper;
    MoveL Offs(pOrigin,78.50,54.78,6.00),v60,z5,tPen\WObj:=wPaper;
    MoveL Offs(pOrigin,77.75,56.89,6.00),vTravel,z5,tPen\WObj:=wPaper;
    MoveL Offs(pOrigin,77.75,56.89,0.00),v60,z0,tPen\WObj:=wPaper;
    MoveL Offs(pOrigin,96.65,56.89,0.00),v40,fine,tPen\WObj:=wPaper;
    MoveL Offs(pOrigin,96.65,56.89,6.00),v60,z5,tPen\WObj:=wPaper;
    MoveL Offs(pOrigin,96.74,59.07,6.00),vTravel,z5,tPen\WObj:=wPaper;
    MoveL Offs(pOrigin,96.74,59.07,0.00),v60,z0,tPen\WObj:=wPaper;
    MoveL Offs(pOrigin,88.36,50.69,0.00),v40,z0,tPen\WObj:=wPaper;
    MoveL Offs(pOrigin,88.88,49.64,0.00),v40,z0,tPen\WObj:=wPaper;
  ENDPROC

  PROC DrawPart12()
    MoveL Offs(pOrigin,73.18,65.34,0.00),v40,fine,tPen\WObj:=wPaper;
    MoveL Offs(pOrigin,73.18,65.34,6.00),v60,z5,tPen\WObj:=wPaper;
    MoveL Offs(pOrigin,75.20,64.28,6.00),vTravel,z5,tPen\WObj:=wPaper;
    MoveL Offs(pOrigin,75.20,64.28,0.00),v60,z0,tPen\WObj:=wPaper;
    MoveL Offs(pOrigin,93.95,64.28,0.00),v40,z0,tPen\WObj:=wPaper;
    MoveL Offs(pOrigin,94.81,64.61,0.00),v40,z0,tPen\WObj:=wPaper;
    MoveL Offs(pOrigin,80.92,50.71,0.00),v40,fine,tPen\WObj:=wPaper;
    MoveL Offs(pOrigin,80.92,50.71,6.00),v60,z5,tPen\WObj:=wPaper;
    MoveL Offs(pOrigin,77.00,59.00,6.00),vTravel,z5,tPen\WObj:=wPaper;
    MoveL Offs(pOrigin,77.00,59.00,0.00),v60,z0,tPen\WObj:=wPaper;
    MoveL Offs(pOrigin,95.90,59.00,0.00),v40,z0,tPen\WObj:=wPaper;
    MoveL Offs(pOrigin,95.60,60.06,0.00),v40,z0,tPen\WObj:=wPaper;
    MoveL Offs(pOrigin,76.70,60.06,0.00),v40,fine,tPen\WObj:=wPaper;
    MoveL Offs(pOrigin,76.70,60.06,6.00),v60,z5,tPen\WObj:=wPaper;
    MoveL Offs(pOrigin,75.65,63.22,6.00),vTravel,z5,tPen\WObj:=wPaper;
    MoveL Offs(pOrigin,75.65,63.22,0.00),v60,z0,tPen\WObj:=wPaper;
    MoveL Offs(pOrigin,94.40,63.22,0.00),v40,fine,tPen\WObj:=wPaper;
    MoveL Offs(pOrigin,94.40,63.22,6.00),v60,z5,tPen\WObj:=wPaper;
    MoveL Offs(pOrigin,105.52,65.86,6.00),vTravel,z5,tPen\WObj:=wPaper;
    MoveL Offs(pOrigin,105.52,65.86,0.00),v60,z0,tPen\WObj:=wPaper;
    MoveL Offs(pOrigin,121.86,49.52,0.00),v40,fine,tPen\WObj:=wPaper;
    MoveL Offs(pOrigin,121.86,49.52,6.00),v60,z5,tPen\WObj:=wPaper;
    MoveL Offs(pOrigin,121.23,50.70,6.00),vTravel,z5,tPen\WObj:=wPaper;
    MoveL Offs(pOrigin,121.23,50.70,0.00),v60,z0,tPen\WObj:=wPaper;
    MoveL Offs(pOrigin,132.05,61.52,0.00),v40,z0,tPen\WObj:=wPaper;
    MoveL Offs(pOrigin,132.84,60.93,0.00),v40,z0,tPen\WObj:=wPaper;
    MoveL Offs(pOrigin,105.90,87.87,0.00),v40,fine,tPen\WObj:=wPaper;
    MoveL Offs(pOrigin,105.90,87.87,6.00),v60,z5,tPen\WObj:=wPaper;
    MoveL Offs(pOrigin,106.23,89.05,6.00),vTravel,z5,tPen\WObj:=wPaper;
    MoveL Offs(pOrigin,106.23,89.05,0.00),v60,z0,tPen\WObj:=wPaper;
    MoveL Offs(pOrigin,132.64,62.63,0.00),v40,z0,tPen\WObj:=wPaper;
    MoveL Offs(pOrigin,131.83,62.80,0.00),v40,z0,tPen\WObj:=wPaper;
    MoveL Offs(pOrigin,119.74,50.71,0.00),v40,z0,tPen\WObj:=wPaper;
    MoveL Offs(pOrigin,120.15,49.73,0.00),v40,z0,tPen\WObj:=wPaper;
    MoveL Offs(pOrigin,106.05,63.84,0.00),v40,z0,tPen\WObj:=wPaper;
    MoveL Offs(pOrigin,106.94,63.30,0.00),v40,z0,tPen\WObj:=wPaper;
    MoveL Offs(pOrigin,132.08,88.43,0.00),v40,z0,tPen\WObj:=wPaper;
    MoveL Offs(pOrigin,131.30,88.57,0.00),v40,z0,tPen\WObj:=wPaper;
    MoveL Offs(pOrigin,107.90,88.57,0.00),v40,z0,tPen\WObj:=wPaper;
    MoveL Offs(pOrigin,106.87,88.61,0.00),v40,z0,tPen\WObj:=wPaper;
    MoveL Offs(pOrigin,109.10,90.84,0.00),v40,fine,tPen\WObj:=wPaper;
    MoveL Offs(pOrigin,109.10,90.84,6.00),v60,z5,tPen\WObj:=wPaper;
    MoveL Offs(pOrigin,110.38,90.62,6.00),vTravel,z5,tPen\WObj:=wPaper;
    MoveL Offs(pOrigin,110.38,90.62,0.00),v60,z0,tPen\WObj:=wPaper;
    MoveL Offs(pOrigin,106.88,87.12,0.00),v40,z0,tPen\WObj:=wPaper;
    MoveL Offs(pOrigin,107.90,87.51,0.00),v40,z0,tPen\WObj:=wPaper;
    MoveL Offs(pOrigin,131.30,87.51,0.00),v40,z0,tPen\WObj:=wPaper;
    MoveL Offs(pOrigin,132.09,86.95,0.00),v40,z0,tPen\WObj:=wPaper;
    MoveL Offs(pOrigin,106.95,61.81,0.00),v40,z0,tPen\WObj:=wPaper;
    MoveL Offs(pOrigin,106.15,62.24,0.00),v40,z0,tPen\WObj:=wPaper;
    MoveL Offs(pOrigin,118.67,49.72,0.00),v40,z0,tPen\WObj:=wPaper;
    MoveL Offs(pOrigin,118.25,50.71,0.00),v40,z0,tPen\WObj:=wPaper;
    MoveL Offs(pOrigin,131.83,64.29,0.00),v40,z0,tPen\WObj:=wPaper;
    MoveL Offs(pOrigin,131.15,64.28,0.00),v40,z0,tPen\WObj:=wPaper;
    MoveL Offs(pOrigin,107.90,64.28,0.00),v40,z0,tPen\WObj:=wPaper;
    MoveL Offs(pOrigin,107.90,65.34,0.00),v40,z0,tPen\WObj:=wPaper;
    MoveL Offs(pOrigin,131.15,65.34,0.00),v40,z0,tPen\WObj:=wPaper;
    MoveL Offs(pOrigin,131.15,66.39,0.00),v40,z0,tPen\WObj:=wPaper;
    MoveL Offs(pOrigin,107.90,66.39,0.00),v40,z0,tPen\WObj:=wPaper;
    MoveL Offs(pOrigin,106.93,66.28,0.00),v40,z0,tPen\WObj:=wPaper;
    MoveL Offs(pOrigin,131.01,90.35,0.00),v40,z0,tPen\WObj:=wPaper;
    MoveL Offs(pOrigin,131.02,91.14,0.00),v40,z0,tPen\WObj:=wPaper;
    MoveL Offs(pOrigin,132.50,89.65,0.00),v40,z0,tPen\WObj:=wPaper;
    MoveL Offs(pOrigin,131.76,89.61,0.00),v40,z0,tPen\WObj:=wPaper;
    MoveL Offs(pOrigin,106.94,64.79,0.00),v40,fine,tPen\WObj:=wPaper;
    MoveL Offs(pOrigin,106.94,64.79,6.00),v60,z5,tPen\WObj:=wPaper;
    MoveL Offs(pOrigin,107.90,63.22,6.00),vTravel,z5,tPen\WObj:=wPaper;
    MoveL Offs(pOrigin,107.90,63.22,0.00),v60,z0,tPen\WObj:=wPaper;
    MoveL Offs(pOrigin,131.15,63.22,0.00),v40,z0,tPen\WObj:=wPaper;
    MoveL Offs(pOrigin,131.15,62.17,0.00),v40,z0,tPen\WObj:=wPaper;
    MoveL Offs(pOrigin,107.90,62.17,0.00),v40,z0,tPen\WObj:=wPaper;
    MoveL Offs(pOrigin,107.90,61.11,0.00),v40,z0,tPen\WObj:=wPaper;
    MoveL Offs(pOrigin,131.15,61.11,0.00),v40,z0,tPen\WObj:=wPaper;
    MoveL Offs(pOrigin,131.15,60.06,0.00),v40,z0,tPen\WObj:=wPaper;
    MoveL Offs(pOrigin,107.90,60.06,0.00),v40,z0,tPen\WObj:=wPaper;
    MoveL Offs(pOrigin,106.95,60.32,0.00),v40,z0,tPen\WObj:=wPaper;
    MoveL Offs(pOrigin,131.88,85.24,0.00),v40,z0,tPen\WObj:=wPaper;
    MoveL Offs(pOrigin,132.59,85.08,0.00),v40,z0,tPen\WObj:=wPaper;
    MoveL Offs(pOrigin,126.76,90.91,0.00),v40,z0,tPen\WObj:=wPaper;
    MoveL Offs(pOrigin,126.65,90.47,0.00),v40,z0,tPen\WObj:=wPaper;
    MoveL Offs(pOrigin,106.92,70.74,0.00),v40,z0,tPen\WObj:=wPaper;
    MoveL Offs(pOrigin,107.90,70.62,0.00),v40,z0,tPen\WObj:=wPaper;
    MoveL Offs(pOrigin,131.15,70.62,0.00),v40,z0,tPen\WObj:=wPaper;
    MoveL Offs(pOrigin,131.81,70.25,0.00),v40,z0,tPen\WObj:=wPaper;
    MoveL Offs(pOrigin,112.30,50.73,0.00),v40,z0,tPen\WObj:=wPaper;
    MoveL Offs(pOrigin,112.71,49.71,0.00),v40,z0,tPen\WObj:=wPaper;
    MoveL Offs(pOrigin,106.13,56.28,0.00),v40,z0,tPen\WObj:=wPaper;
    MoveL Offs(pOrigin,106.96,55.85,0.00),v40,z0,tPen\WObj:=wPaper;
    MoveL Offs(pOrigin,131.89,80.78,0.00),v40,z0,tPen\WObj:=wPaper;
    MoveL Offs(pOrigin,132.58,80.61,0.00),v40,z0,tPen\WObj:=wPaper;
    MoveL Offs(pOrigin,105.75,107.45,0.00),v40,z0,tPen\WObj:=wPaper;
    MoveL Offs(pOrigin,106.82,107.97,0.00),v40,z0,tPen\WObj:=wPaper;
    MoveL Offs(pOrigin,131.74,132.90,0.00),v40,z0,tPen\WObj:=wPaper;
    MoveL Offs(pOrigin,132.05,133.18,0.00),v40,z0,tPen\WObj:=wPaper;
    MoveL Offs(pOrigin,107.75,133.27,0.00),v40,z0,tPen\WObj:=wPaper;
    MoveL Offs(pOrigin,107.05,132.98,0.00),v40,z0,tPen\WObj:=wPaper;
    MoveL Offs(pOrigin,107.00,93.38,0.00),v40,z0,tPen\WObj:=wPaper;
    MoveL Offs(pOrigin,107.30,92.97,0.00),v40,z0,tPen\WObj:=wPaper;
    MoveL Offs(pOrigin,132.15,93.07,0.00),v40,z0,tPen\WObj:=wPaper;
    MoveL Offs(pOrigin,132.05,133.18,0.00),v40,z0,tPen\WObj:=wPaper;
    MoveL Offs(pOrigin,132.84,132.63,0.00),v40,z0,tPen\WObj:=wPaper;
    MoveL Offs(pOrigin,131.46,134.00,0.00),v40,z0,tPen\WObj:=wPaper;
    MoveL Offs(pOrigin,130.68,133.33,0.00),v40,z0,tPen\WObj:=wPaper;
    MoveL Offs(pOrigin,106.92,109.57,0.00),v40,z0,tPen\WObj:=wPaper;
    MoveL Offs(pOrigin,107.75,109.69,0.00),v40,z0,tPen\WObj:=wPaper;
    MoveL Offs(pOrigin,131.30,109.69,0.00),v40,z0,tPen\WObj:=wPaper;
    MoveL Offs(pOrigin,132.02,109.28,0.00),v40,z0,tPen\WObj:=wPaper;
    MoveL Offs(pOrigin,115.69,92.95,0.00),v40,fine,tPen\WObj:=wPaper;
    MoveL Offs(pOrigin,115.69,92.95,6.00),v60,z5,tPen\WObj:=wPaper;
    MoveL Offs(pOrigin,117.18,92.94,6.00),vTravel,z5,tPen\WObj:=wPaper;
    MoveL Offs(pOrigin,117.18,92.94,0.00),v60,z0,tPen\WObj:=wPaper;
    MoveL Offs(pOrigin,132.03,107.79,0.00),v40,z0,tPen\WObj:=wPaper;
    MoveL Offs(pOrigin,131.30,107.58,0.00),v40,z0,tPen\WObj:=wPaper;
    MoveL Offs(pOrigin,107.75,107.58,0.00),v40,z0,tPen\WObj:=wPaper;
    MoveL Offs(pOrigin,107.75,108.63,0.00),v40,z0,tPen\WObj:=wPaper;
    MoveL Offs(pOrigin,131.30,108.63,0.00),v40,fine,tPen\WObj:=wPaper;
    MoveL Offs(pOrigin,131.30,108.63,6.00),v60,z5,tPen\WObj:=wPaper;
    MoveL Offs(pOrigin,132.77,108.80,6.00),vTravel,z5,tPen\WObj:=wPaper;
    MoveL Offs(pOrigin,132.77,108.80,0.00),v60,z0,tPen\WObj:=wPaper;
    MoveL Offs(pOrigin,107.63,133.94,0.00),v40,z0,tPen\WObj:=wPaper;
  ENDPROC

